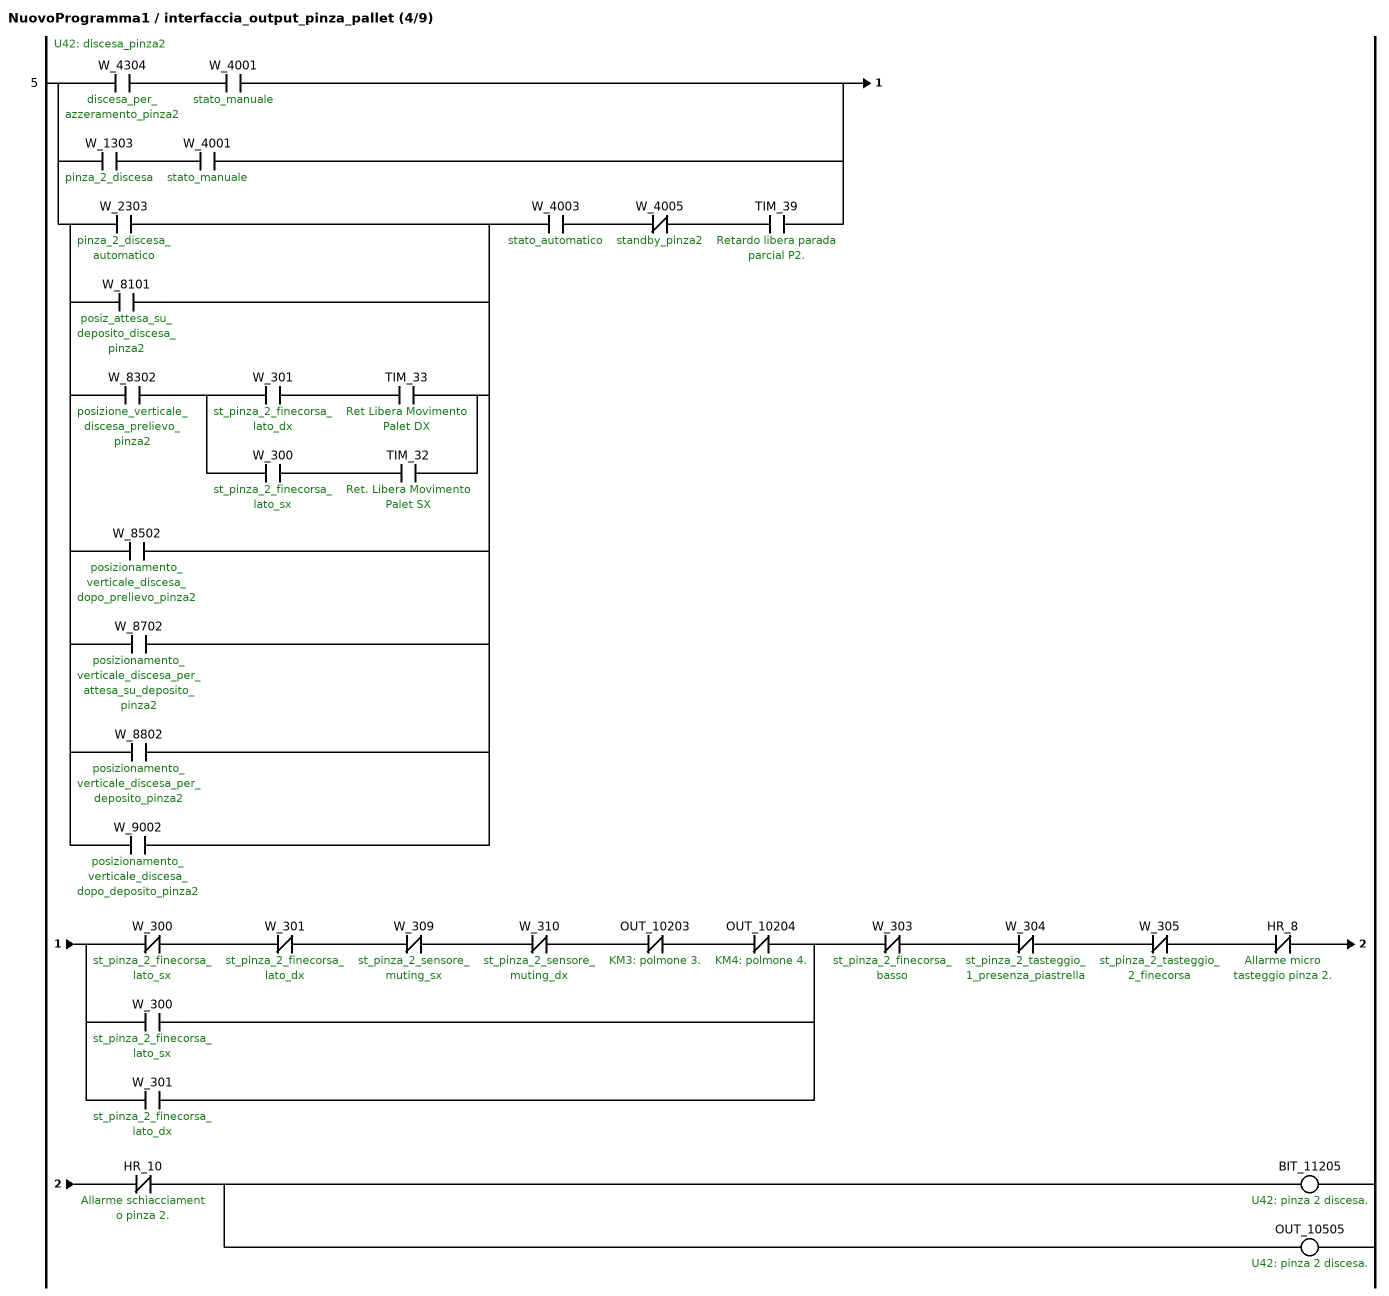
; [picture p24: NuovoProgramma1 / interfaccia_output_pinza_pallet, rungs 5-5]
; rung 5: U42: discesa_pinza2
LD W_4304  ; discesa_per_azzeramento_pinza2
AND W_4001  ; stato_manuale
LD W_1303  ; pinza_2_discesa
AND W_4001  ; stato_manuale
ORLD
LD W_2303  ; pinza_2_discesa_automatico
OR W_8101  ; posiz_attesa_su_deposito_discesa_pinza2
LD W_8302  ; posizione_verticale_discesa_prelievo_pinza2
LD W_301  ; st_pinza_2_finecorsa_lato_dx
AND TIM_33  ; Ret Libera Movimento Palet DX
LD W_300  ; st_pinza_2_finecorsa_lato_sx
AND TIM_32  ; Ret. Libera Movimento Palet SX
ORLD
ANDLD
ORLD
OR W_8502  ; posizionamento_verticale_discesa_dopo_prelievo_pinza2
OR W_8702  ; posizionamento_verticale_discesa_per_attesa_su_deposito_pinza2
OR W_8802  ; posizionamento_verticale_discesa_per_deposito_pinza2
OR W_9002  ; posizionamento_verticale_discesa_dopo_deposito_pinza2
AND W_4003  ; stato_automatico
ANDNOT W_4005  ; standby_pinza2
AND TIM_39  ; Retardo libera parada parcial P2.
ORLD
LDNOT W_300  ; st_pinza_2_finecorsa_lato_sx
ANDNOT W_301  ; st_pinza_2_finecorsa_lato_dx
ANDNOT W_309  ; st_pinza_2_sensore_muting_sx
ANDNOT W_310  ; st_pinza_2_sensore_muting_dx
ANDNOT OUT_10203  ; KM3: polmone 3.
ANDNOT OUT_10204  ; KM4: polmone 4.
OR W_300  ; st_pinza_2_finecorsa_lato_sx
OR W_301  ; st_pinza_2_finecorsa_lato_dx
ANDLD
ANDNOT W_303  ; st_pinza_2_finecorsa_basso
ANDNOT W_304  ; st_pinza_2_tasteggio_1_presenza_piastrella
ANDNOT W_305  ; st_pinza_2_tasteggio_2_finecorsa
ANDNOT HR_8  ; Allarme micro tasteggio pinza 2.
ANDNOT HR_10  ; Allarme schiacciamento pinza 2.
OUT BIT_11205  ; U42: pinza 2 discesa.
OUT OUT_10505  ; U42: pinza 2 discesa.

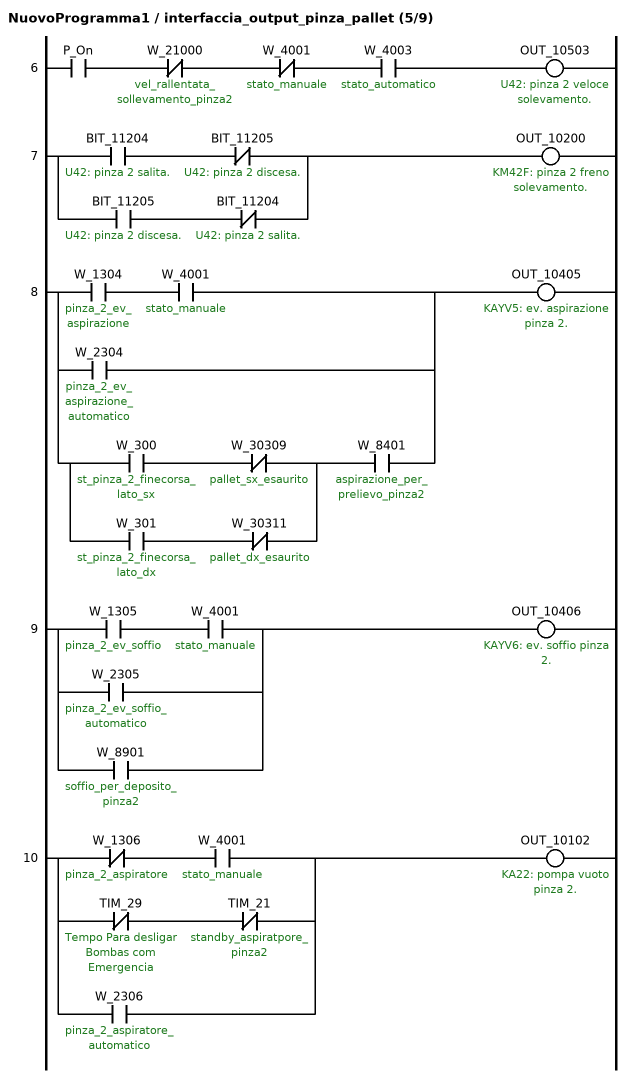
; rung 6
LD P_On
ANDNOT W_21000  ; vel_rallentata_sollevamento_pinza2
ANDNOT W_4001  ; stato_manuale
AND W_4003  ; stato_automatico
OUT OUT_10503  ; U42: pinza 2 veloce solevamento.
; rung 7
LD BIT_11204  ; U42: pinza 2 salita.
ANDNOT BIT_11205  ; U42: pinza 2 discesa.
LD BIT_11205  ; U42: pinza 2 discesa.
ANDNOT BIT_11204  ; U42: pinza 2 salita.
ORLD
OUT OUT_10200  ; KM42F: pinza 2 freno solevamento.
; rung 8
LD W_1304  ; pinza_2_ev_aspirazione
AND W_4001  ; stato_manuale
OR W_2304  ; pinza_2_ev_aspirazione_automatico
LD W_300  ; st_pinza_2_finecorsa_lato_sx
ANDNOT W_30309  ; pallet_sx_esaurito
LD W_301  ; st_pinza_2_finecorsa_lato_dx
ANDNOT W_30311  ; pallet_dx_esaurito
ORLD
AND W_8401  ; aspirazione_per_prelievo_pinza2
ORLD
OUT OUT_10405  ; KAYV5: ev. aspirazione pinza 2.
; rung 9
LD W_1305  ; pinza_2_ev_soffio
AND W_4001  ; stato_manuale
OR W_2305  ; pinza_2_ev_soffio_automatico
OR W_8901  ; soffio_per_deposito_pinza2
OUT OUT_10406  ; KAYV6: ev. soffio pinza 2.
; rung 10
LDNOT W_1306  ; pinza_2_aspiratore
AND W_4001  ; stato_manuale
LDNOT TIM_29  ; Tempo Para desligar Bombas com Emergencia
ANDNOT TIM_21  ; standby_aspiratpore_pinza2
ORLD
OR W_2306  ; pinza_2_aspiratore_automatico
OUT OUT_10102  ; KA22: pompa vuoto pinza 2.

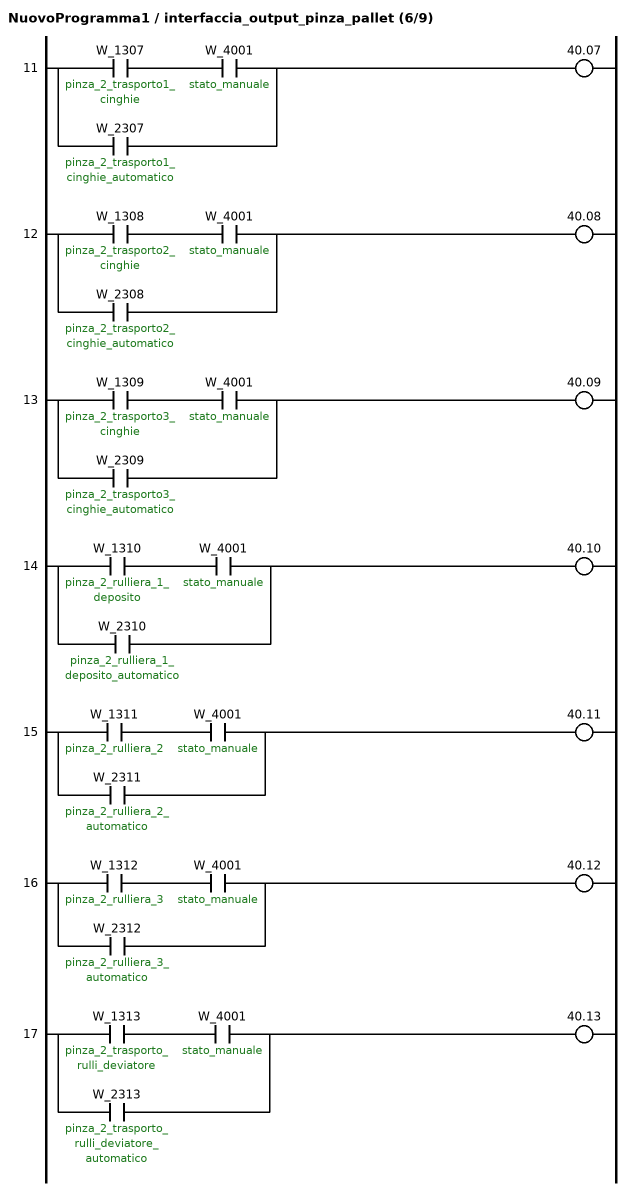
; rung 11
LD W_1307  ; pinza_2_trasporto1_cinghie
AND W_4001  ; stato_manuale
OR W_2307  ; pinza_2_trasporto1_cinghie_automatico
OUT 40.07
; rung 12
LD W_1308  ; pinza_2_trasporto2_cinghie
AND W_4001  ; stato_manuale
OR W_2308  ; pinza_2_trasporto2_cinghie_automatico
OUT 40.08
; rung 13
LD W_1309  ; pinza_2_trasporto3_cinghie
AND W_4001  ; stato_manuale
OR W_2309  ; pinza_2_trasporto3_cinghie_automatico
OUT 40.09
; rung 14
LD W_1310  ; pinza_2_rulliera_1_deposito
AND W_4001  ; stato_manuale
OR W_2310  ; pinza_2_rulliera_1_deposito_automatico
OUT 40.10
; rung 15
LD W_1311  ; pinza_2_rulliera_2
AND W_4001  ; stato_manuale
OR W_2311  ; pinza_2_rulliera_2_automatico
OUT 40.11
; rung 16
LD W_1312  ; pinza_2_rulliera_3
AND W_4001  ; stato_manuale
OR W_2312  ; pinza_2_rulliera_3_automatico
OUT 40.12
; rung 17
LD W_1313  ; pinza_2_trasporto_rulli_deviatore
AND W_4001  ; stato_manuale
OR W_2313  ; pinza_2_trasporto_rulli_deviatore_automatico
OUT 40.13

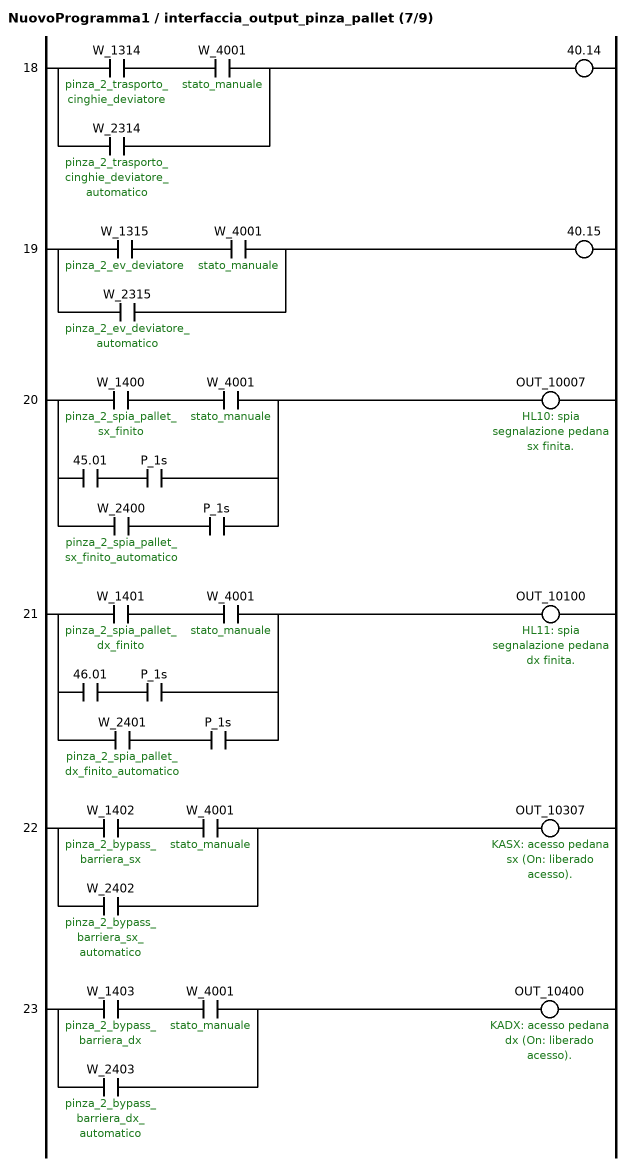
; rung 18
LD W_1314  ; pinza_2_trasporto_cinghie_deviatore
AND W_4001  ; stato_manuale
OR W_2314  ; pinza_2_trasporto_cinghie_deviatore_automatico
OUT 40.14
; rung 19
LD W_1315  ; pinza_2_ev_deviatore
AND W_4001  ; stato_manuale
OR W_2315  ; pinza_2_ev_deviatore_automatico
OUT 40.15
; rung 20
LD W_1400  ; pinza_2_spia_pallet_sx_finito
AND W_4001  ; stato_manuale
LD 45.01
AND P_1s
ORLD
LD W_2400  ; pinza_2_spia_pallet_sx_finito_automatico
AND P_1s
ORLD
OUT OUT_10007  ; HL10: spia segnalazione pedana sx finita.
; rung 21
LD W_1401  ; pinza_2_spia_pallet_dx_finito
AND W_4001  ; stato_manuale
LD 46.01
AND P_1s
ORLD
LD W_2401  ; pinza_2_spia_pallet_dx_finito_automatico
AND P_1s
ORLD
OUT OUT_10100  ; HL11: spia segnalazione pedana dx finita.
; rung 22
LD W_1402  ; pinza_2_bypass_barriera_sx
AND W_4001  ; stato_manuale
OR W_2402  ; pinza_2_bypass_barriera_sx_automatico
OUT OUT_10307  ; KASX: acesso pedana sx (On: liberado acesso).
; rung 23
LD W_1403  ; pinza_2_bypass_barriera_dx
AND W_4001  ; stato_manuale
OR W_2403  ; pinza_2_bypass_barriera_dx_automatico
OUT OUT_10400  ; KADX: acesso pedana dx (On: liberado acesso).

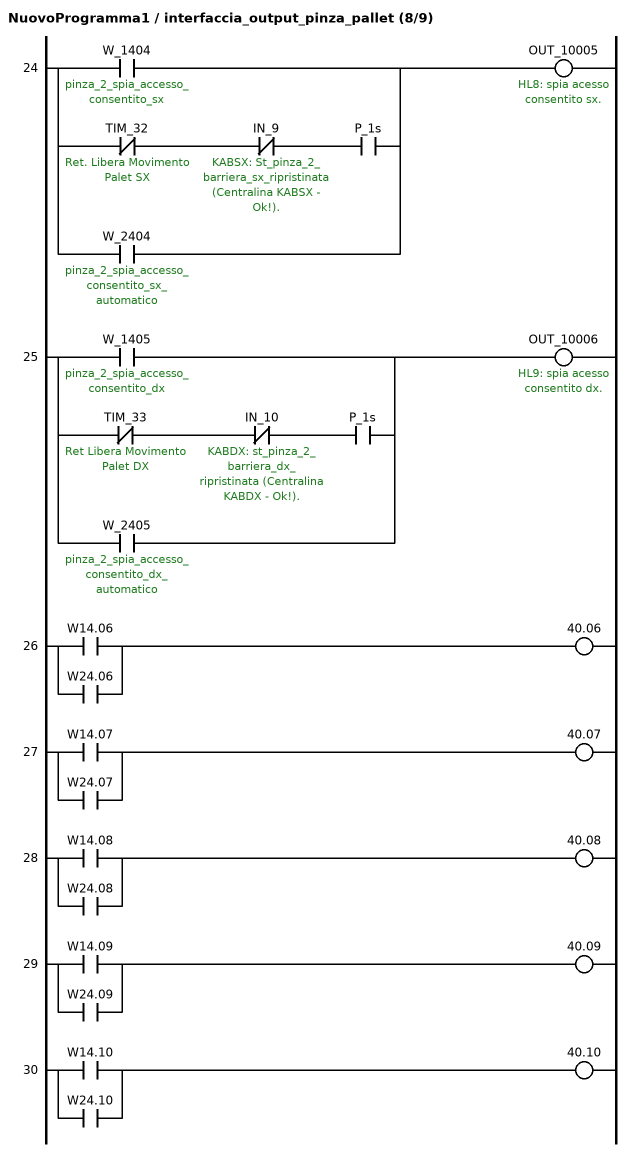
; rung 24
LD W_1404  ; pinza_2_spia_accesso_consentito_sx
LDNOT TIM_32  ; Ret. Libera Movimento Palet SX
ANDNOT IN_9  ; KABSX: St_pinza_2_barriera_sx_ripristinata (Centralina KABSX - Ok!).
AND P_1s
ORLD
OR W_2404  ; pinza_2_spia_accesso_consentito_sx_automatico
OUT OUT_10005  ; HL8: spia acesso consentito sx.
; rung 25
LD W_1405  ; pinza_2_spia_accesso_consentito_dx
LDNOT TIM_33  ; Ret Libera Movimento Palet DX
ANDNOT IN_10  ; KABDX: st_pinza_2_barriera_dx_ripristinata (Centralina KABDX - Ok!).
AND P_1s
ORLD
OR W_2405  ; pinza_2_spia_accesso_consentito_dx_automatico
OUT OUT_10006  ; HL9: spia acesso consentito dx.
; rung 26
LD W14.06
OR W24.06
OUT 40.06
; rung 27
LD W14.07
OR W24.07
OUT 40.07
; rung 28
LD W14.08
OR W24.08
OUT 40.08
; rung 29
LD W14.09
OR W24.09
OUT 40.09
; rung 30
LD W14.10
OR W24.10
OUT 40.10

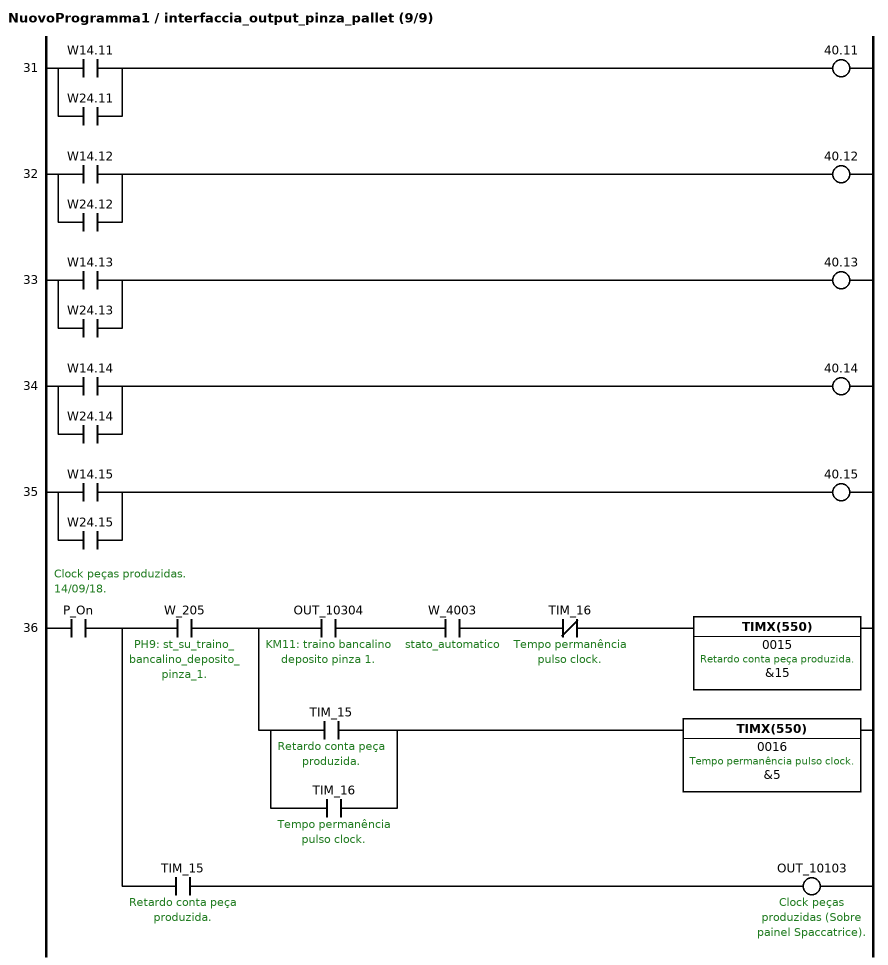
; rung 31
LD W14.11
OR W24.11
OUT 40.11
; rung 32
LD W14.12
OR W24.12
OUT 40.12
; rung 33
LD W14.13
OR W24.13
OUT 40.13
; rung 34
LD W14.14
OR W24.14
OUT 40.14
; rung 35
LD W14.15
OR W24.15
OUT 40.15
; rung 36: Clock peças produzidas. / 14/09/18.
LD P_On
OUT TR0
AND W_205  ; PH9: st_su_traino_bancalino_deposito_pinza_1.
OUT TR1
AND OUT_10304  ; KM11: traino bancalino deposito pinza 1.
AND W_4003  ; stato_automatico
ANDNOT TIM_16  ; Tempo permanência pulso clock.
TIMX(550) 0015 &15  ; Retardo conta peça produzida.
LD TR1
LD TIM_15  ; Retardo conta peça produzida.
OR TIM_16  ; Tempo permanência pulso clock.
ANDLD
TIMX(550) 0016 &5  ; Tempo permanência pulso clock.
LD TR0
AND TIM_15  ; Retardo conta peça produzida.
OUT OUT_10103  ; Clock peças produzidas (Sobre painel Spaccatrice).

### Section manuale

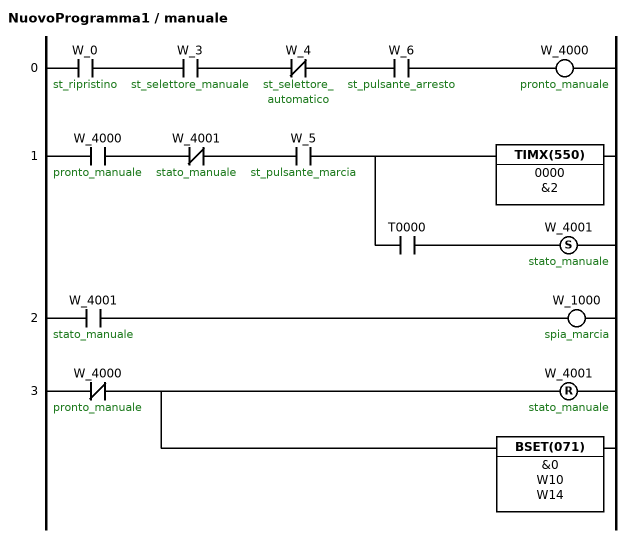
; rung 0
LD W_0  ; st_ripristino
AND W_3  ; st_selettore_manuale
ANDNOT W_4  ; st_selettore_automatico
AND W_6  ; st_pulsante_arresto
OUT W_4000  ; pronto_manuale
; rung 1
LD W_4000  ; pronto_manuale
ANDNOT W_4001  ; stato_manuale
AND W_5  ; st_pulsante_marcia
TIMX(550) 0000 &2
AND T0000
SET W_4001  ; stato_manuale
; rung 2
LD W_4001  ; stato_manuale
OUT W_1000  ; spia_marcia
; rung 3
LDNOT W_4000  ; pronto_manuale
RSET W_4001  ; stato_manuale
BSET(071) &0 W10 W14

### Section abilitazioni

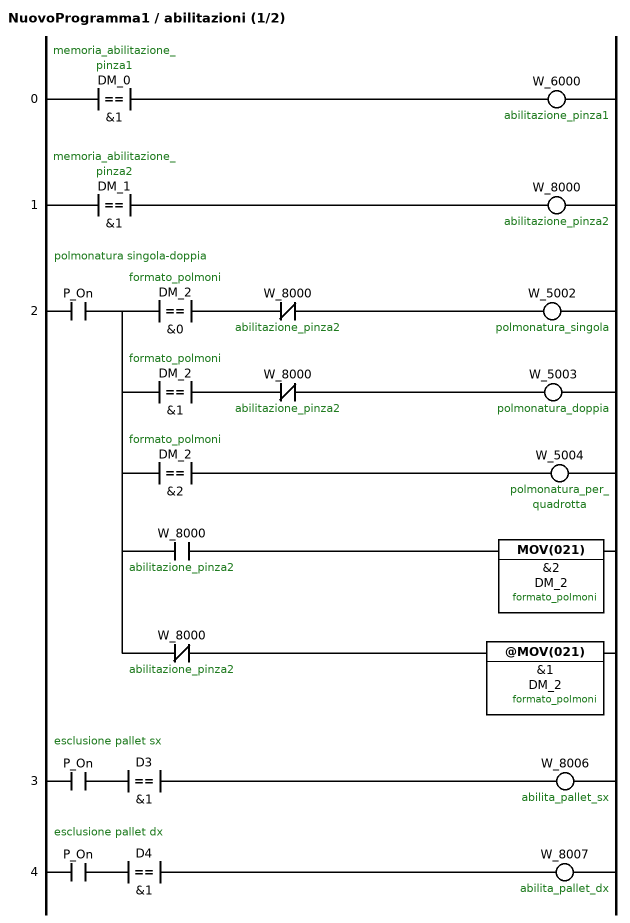
; rung 0
LD=(300) DM_0 &1  ; memoria_abilitazione_pinza1
OUT W_6000  ; abilitazione_pinza1
; rung 1
LD=(300) DM_1 &1  ; memoria_abilitazione_pinza2
OUT W_8000  ; abilitazione_pinza2
; rung 2: polmonatura singola-doppia
LD P_On
OUT TR0
AND=(300) DM_2 &0  ; formato_polmoni
ANDNOT W_8000  ; abilitazione_pinza2
OUT W_5002  ; polmonatura_singola
LD TR0
AND=(300) DM_2 &1  ; formato_polmoni
ANDNOT W_8000  ; abilitazione_pinza2
OUT W_5003  ; polmonatura_doppia
LD TR0
AND=(300) DM_2 &2  ; formato_polmoni
OUT W_5004  ; polmonatura_per_quadrotta
LD TR0
AND W_8000  ; abilitazione_pinza2
MOV(021) &2 DM_2  ; formato_polmoni
LD TR0
ANDNOT W_8000  ; abilitazione_pinza2
@MOV(021) &1 DM_2  ; formato_polmoni
; rung 3: esclusione pallet sx
LD P_On
AND=(300) D3 &1
OUT W_8006  ; abilita_pallet_sx
; rung 4: esclusione pallet dx
LD P_On
AND=(300) D4 &1
OUT W_8007  ; abilita_pallet_dx

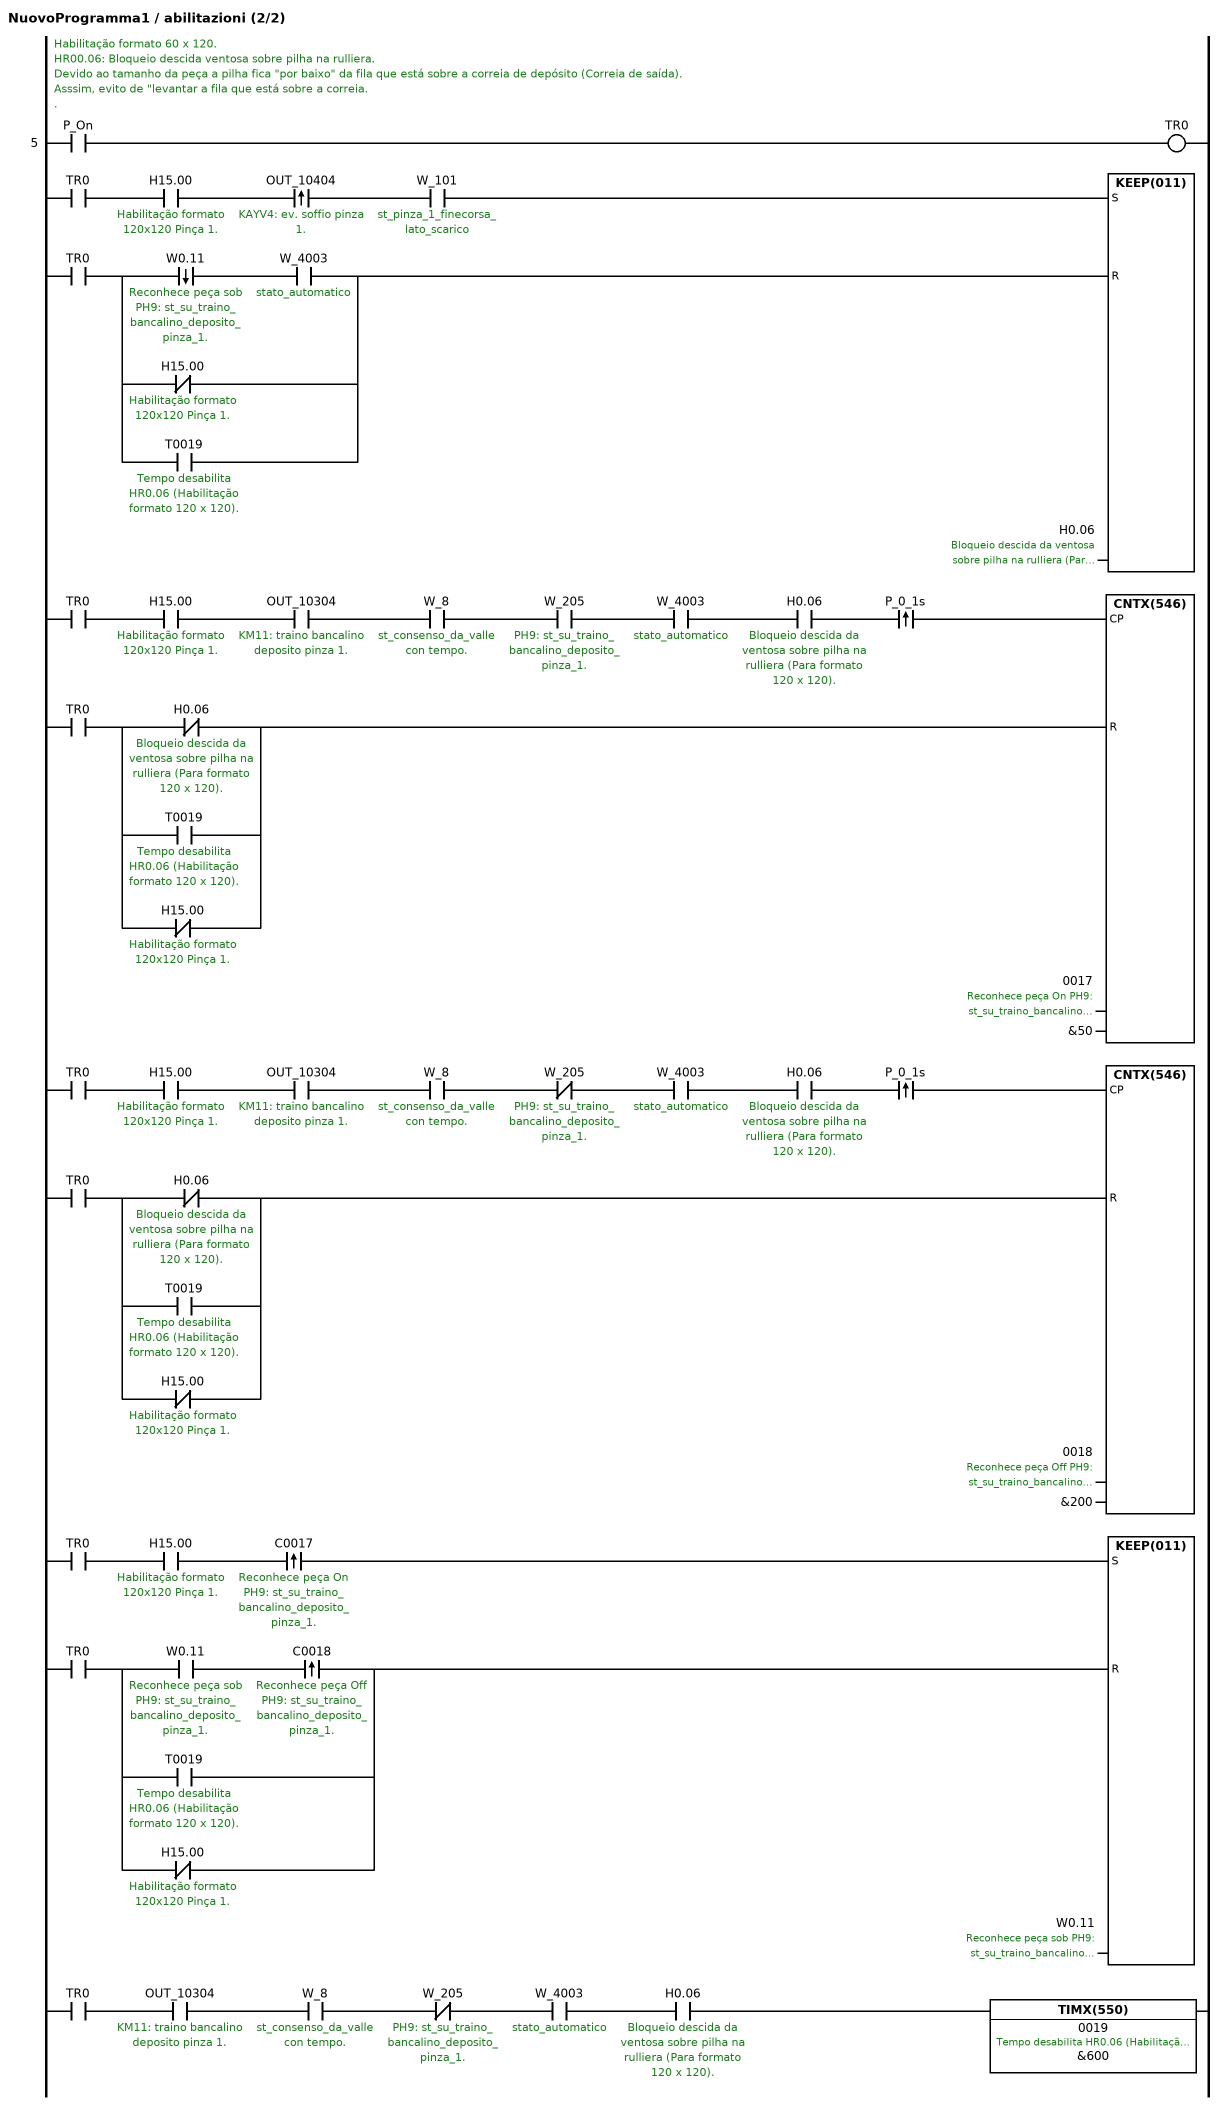
; rung 5: Habilitação formato 60 x 120. / HR00.06: Bloqueio descida ventosa sobre pilha na rulliera. / Devido ao tamanho da peça a pilha fica "por baixo" da fila que está sobre a correia de depósito (Correia de saída). / Asssim, evito de "levantar a fila que está sobre a correia. / .
LD P_On
OUT TR0
AND H15.00  ; Habilitação formato 120x120 Pinça 1.
@AND OUT_10404  ; KAYV4: ev. soffio pinza 1.
AND W_101  ; st_pinza_1_finecorsa_lato_scarico
LD TR0
%LD W0.11  ; Reconhece peça sob PH9: st_su_traino_bancalino_deposito_pinza_1.
AND W_4003  ; stato_automatico
ORNOT H15.00  ; Habilitação formato 120x120 Pinça 1.
OR T0019  ; Tempo desabilita HR0.06 (Habilitação formato 120 x 120).
ANDLD
KEEP(011) H0.06  ; Bloqueio descida da ventosa sobre pilha na rulliera (Para formato 120 x 120).  // On: material depositado sobre correia de saída. / Off: passou peça sob Ftc se saída (IN2.09_PH9: st_su_traino_bancalino_deposito_pinza_1). / .
LD TR0
AND H15.00  ; Habilitação formato 120x120 Pinça 1.
AND OUT_10304  ; KM11: traino bancalino deposito pinza 1.
AND W_8  ; st_consenso_da_valle con tempo.
AND W_205  ; PH9: st_su_traino_bancalino_deposito_pinza_1.
AND W_4003  ; stato_automatico
AND H0.06  ; Bloqueio descida da ventosa sobre pilha na rulliera (Para formato 120 x 120).
@AND P_0_1s
LD TR0
LDNOT H0.06  ; Bloqueio descida da ventosa sobre pilha na rulliera (Para formato 120 x 120).
OR T0019  ; Tempo desabilita HR0.06 (Habilitação formato 120 x 120).
ORNOT H15.00  ; Habilitação formato 120x120 Pinça 1.
ANDLD
CNTX(546) 0017 &50  ; Reconhece peça On PH9: st_su_traino_bancalino_deposito_pinza_1.
LD TR0
AND H15.00  ; Habilitação formato 120x120 Pinça 1.
AND OUT_10304  ; KM11: traino bancalino deposito pinza 1.
AND W_8  ; st_consenso_da_valle con tempo.
ANDNOT W_205  ; PH9: st_su_traino_bancalino_deposito_pinza_1.
AND W_4003  ; stato_automatico
AND H0.06  ; Bloqueio descida da ventosa sobre pilha na rulliera (Para formato 120 x 120).
@AND P_0_1s
LD TR0
LDNOT H0.06  ; Bloqueio descida da ventosa sobre pilha na rulliera (Para formato 120 x 120).
OR T0019  ; Tempo desabilita HR0.06 (Habilitação formato 120 x 120).
ORNOT H15.00  ; Habilitação formato 120x120 Pinça 1.
ANDLD
CNTX(546) 0018 &200  ; Reconhece peça Off PH9: st_su_traino_bancalino_deposito_pinza_1.
LD TR0
AND H15.00  ; Habilitação formato 120x120 Pinça 1.
@AND C0017  ; Reconhece peça On PH9: st_su_traino_bancalino_deposito_pinza_1.
LD TR0
LD W0.11  ; Reconhece peça sob PH9: st_su_traino_bancalino_deposito_pinza_1.
@AND C0018  ; Reconhece peça Off PH9: st_su_traino_bancalino_deposito_pinza_1.
OR T0019  ; Tempo desabilita HR0.06 (Habilitação formato 120 x 120).
ORNOT H15.00  ; Habilitação formato 120x120 Pinça 1.
ANDLD
KEEP(011) W0.11  ; Reconhece peça sob PH9: st_su_traino_bancalino_deposito_pinza_1.
LD TR0
AND OUT_10304  ; KM11: traino bancalino deposito pinza 1.
AND W_8  ; st_consenso_da_valle con tempo.
ANDNOT W_205  ; PH9: st_su_traino_bancalino_deposito_pinza_1.
AND W_4003  ; stato_automatico
AND H0.06  ; Bloqueio descida da ventosa sobre pilha na rulliera (Para formato 120 x 120).
TIMX(550) 0019 &600  ; Tempo desabilita HR0.06 (Habilitação formato 120 x 120).  // Tempo de segurança para o caso de faltar material na linha (E, assim, não acionar a ftc. que reconhece passagem da peça). / .

### Section azzeramento_assi_pinza_ribaltino

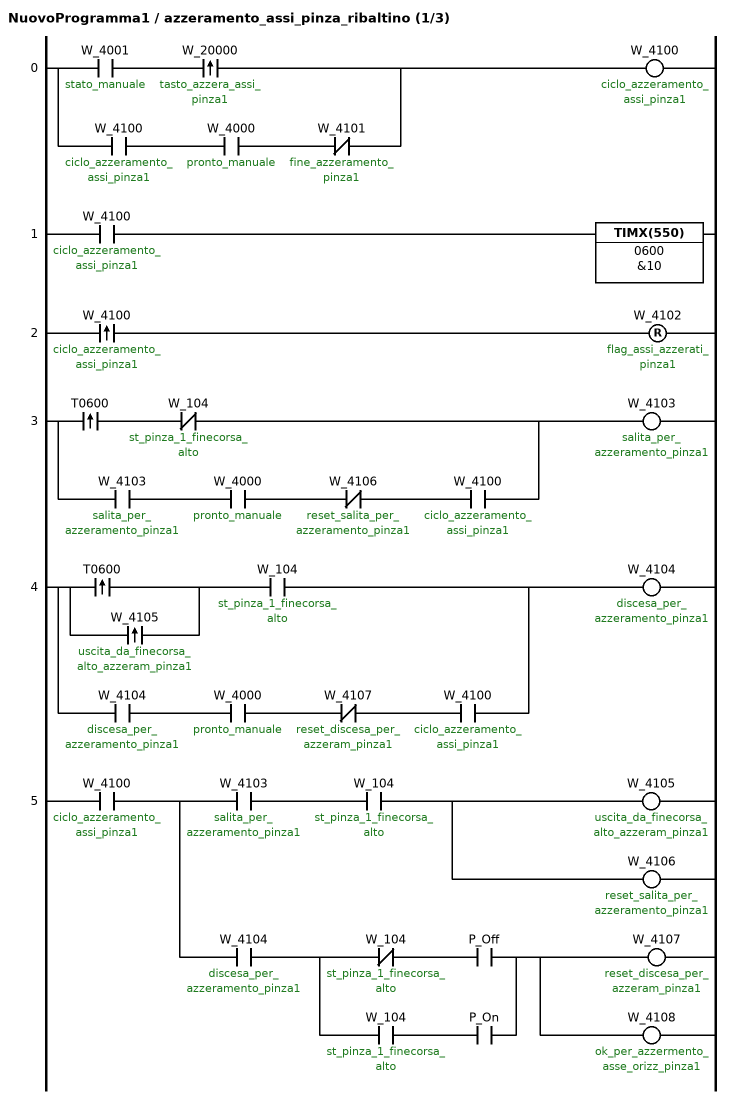
; rung 0
LD W_4001  ; stato_manuale
@AND W_20000  ; tasto_azzera_assi_pinza1
LD W_4100  ; ciclo_azzeramento_assi_pinza1
AND W_4000  ; pronto_manuale
ANDNOT W_4101  ; fine_azzeramento_pinza1
ORLD
OUT W_4100  ; ciclo_azzeramento_assi_pinza1
; rung 1
LD W_4100  ; ciclo_azzeramento_assi_pinza1
TIMX(550) 0600 &10
; rung 2
@LD W_4100  ; ciclo_azzeramento_assi_pinza1
RSET W_4102  ; flag_assi_azzerati_pinza1
; rung 3
@LD T0600
ANDNOT W_104  ; st_pinza_1_finecorsa_alto
LD W_4103  ; salita_per_azzeramento_pinza1
AND W_4000  ; pronto_manuale
ANDNOT W_4106  ; reset_salita_per_azzeramento_pinza1
AND W_4100  ; ciclo_azzeramento_assi_pinza1
ORLD
OUT W_4103  ; salita_per_azzeramento_pinza1
; rung 4
@LD T0600
@OR W_4105  ; uscita_da_finecorsa_alto_azzeram_pinza1
AND W_104  ; st_pinza_1_finecorsa_alto
LD W_4104  ; discesa_per_azzeramento_pinza1
AND W_4000  ; pronto_manuale
ANDNOT W_4107  ; reset_discesa_per_azzeram_pinza1
AND W_4100  ; ciclo_azzeramento_assi_pinza1
ORLD
OUT W_4104  ; discesa_per_azzeramento_pinza1
; rung 5
LD W_4100  ; ciclo_azzeramento_assi_pinza1
OUT TR0
AND W_4103  ; salita_per_azzeramento_pinza1
AND W_104  ; st_pinza_1_finecorsa_alto
OUT W_4105  ; uscita_da_finecorsa_alto_azzeram_pinza1
OUT W_4106  ; reset_salita_per_azzeramento_pinza1
LD TR0
AND W_4104  ; discesa_per_azzeramento_pinza1
LDNOT W_104  ; st_pinza_1_finecorsa_alto
AND P_Off
LD W_104  ; st_pinza_1_finecorsa_alto
AND P_On
ORLD
ANDLD
OUT W_4107  ; reset_discesa_per_azzeram_pinza1
OUT W_4108  ; ok_per_azzermento_asse_orizz_pinza1

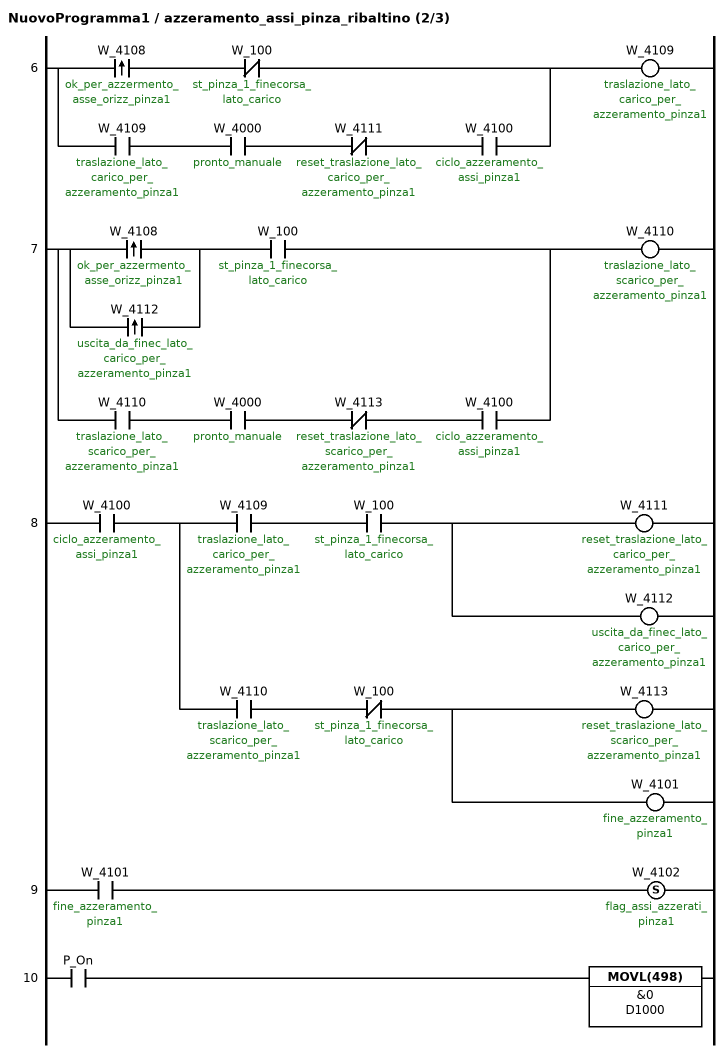
; rung 6
@LD W_4108  ; ok_per_azzermento_asse_orizz_pinza1
ANDNOT W_100  ; st_pinza_1_finecorsa_lato_carico
LD W_4109  ; traslazione_lato_carico_per_azzeramento_pinza1
AND W_4000  ; pronto_manuale
ANDNOT W_4111  ; reset_traslazione_lato_carico_per_azzeramento_pinza1
AND W_4100  ; ciclo_azzeramento_assi_pinza1
ORLD
OUT W_4109  ; traslazione_lato_carico_per_azzeramento_pinza1
; rung 7
@LD W_4108  ; ok_per_azzermento_asse_orizz_pinza1
@OR W_4112  ; uscita_da_finec_lato_carico_per_azzeramento_pinza1
AND W_100  ; st_pinza_1_finecorsa_lato_carico
LD W_4110  ; traslazione_lato_scarico_per_azzeramento_pinza1
AND W_4000  ; pronto_manuale
ANDNOT W_4113  ; reset_traslazione_lato_scarico_per_azzeramento_pinza1
AND W_4100  ; ciclo_azzeramento_assi_pinza1
ORLD
OUT W_4110  ; traslazione_lato_scarico_per_azzeramento_pinza1
; rung 8
LD W_4100  ; ciclo_azzeramento_assi_pinza1
OUT TR0
AND W_4109  ; traslazione_lato_carico_per_azzeramento_pinza1
AND W_100  ; st_pinza_1_finecorsa_lato_carico
OUT W_4111  ; reset_traslazione_lato_carico_per_azzeramento_pinza1
OUT W_4112  ; uscita_da_finec_lato_carico_per_azzeramento_pinza1
LD TR0
AND W_4110  ; traslazione_lato_scarico_per_azzeramento_pinza1
ANDNOT W_100  ; st_pinza_1_finecorsa_lato_carico
OUT W_4113  ; reset_traslazione_lato_scarico_per_azzeramento_pinza1
OUT W_4101  ; fine_azzeramento_pinza1
; rung 9
LD W_4101  ; fine_azzeramento_pinza1
SET W_4102  ; flag_assi_azzerati_pinza1
; rung 10
LD P_On
MOVL(498) &0 D1000

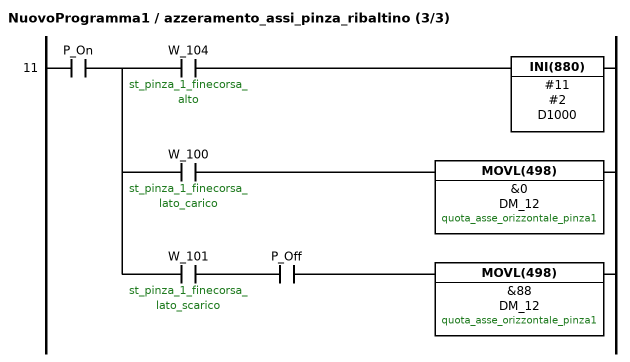
; rung 11
LD P_On
OUT TR0
AND W_104  ; st_pinza_1_finecorsa_alto
INI(880) #11 #2 D1000
LD TR0
AND W_100  ; st_pinza_1_finecorsa_lato_carico
MOVL(498) &0 DM_12  ; quota_asse_orizzontale_pinza1
LD TR0
AND W_101  ; st_pinza_1_finecorsa_lato_scarico
AND P_Off
MOVL(498) &88 DM_12  ; quota_asse_orizzontale_pinza1

### Section azzeramento_assi_pinza_pallet

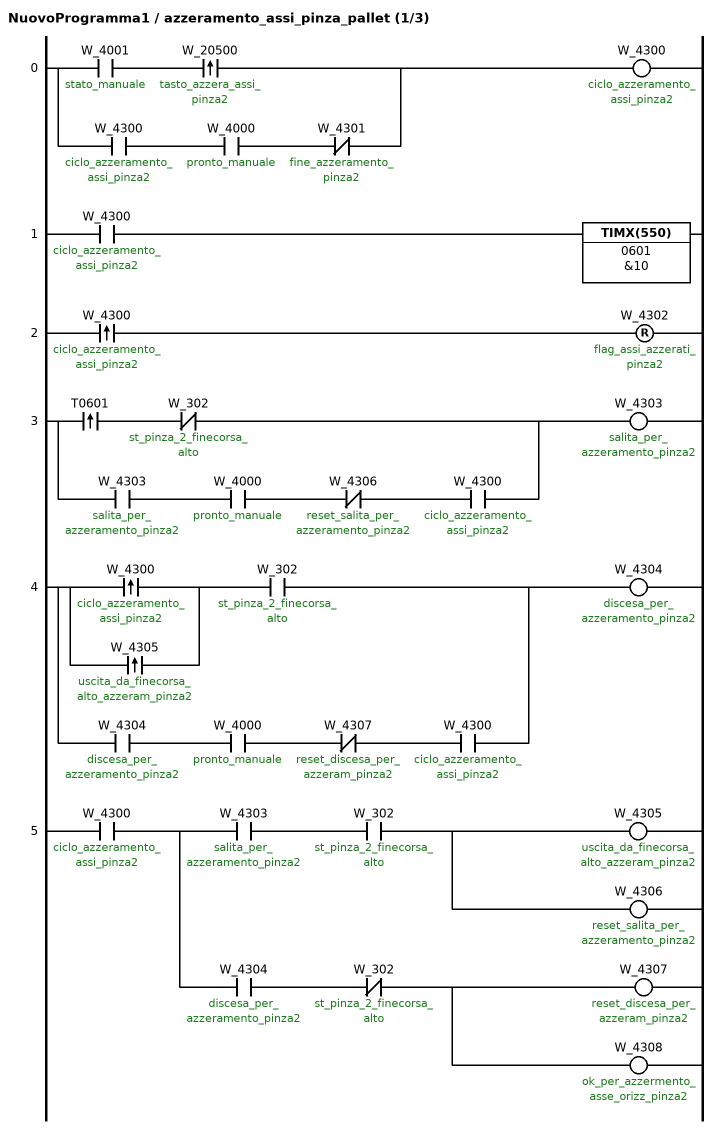
; rung 0
LD W_4001  ; stato_manuale
@AND W_20500  ; tasto_azzera_assi_pinza2
LD W_4300  ; ciclo_azzeramento_assi_pinza2
AND W_4000  ; pronto_manuale
ANDNOT W_4301  ; fine_azzeramento_pinza2
ORLD
OUT W_4300  ; ciclo_azzeramento_assi_pinza2
; rung 1
LD W_4300  ; ciclo_azzeramento_assi_pinza2
TIMX(550) 0601 &10
; rung 2
@LD W_4300  ; ciclo_azzeramento_assi_pinza2
RSET W_4302  ; flag_assi_azzerati_pinza2
; rung 3
@LD T0601
ANDNOT W_302  ; st_pinza_2_finecorsa_alto
LD W_4303  ; salita_per_azzeramento_pinza2
AND W_4000  ; pronto_manuale
ANDNOT W_4306  ; reset_salita_per_azzeramento_pinza2
AND W_4300  ; ciclo_azzeramento_assi_pinza2
ORLD
OUT W_4303  ; salita_per_azzeramento_pinza2
; rung 4
@LD W_4300  ; ciclo_azzeramento_assi_pinza2
@OR W_4305  ; uscita_da_finecorsa_alto_azzeram_pinza2
AND W_302  ; st_pinza_2_finecorsa_alto
LD W_4304  ; discesa_per_azzeramento_pinza2
AND W_4000  ; pronto_manuale
ANDNOT W_4307  ; reset_discesa_per_azzeram_pinza2
AND W_4300  ; ciclo_azzeramento_assi_pinza2
ORLD
OUT W_4304  ; discesa_per_azzeramento_pinza2
; rung 5
LD W_4300  ; ciclo_azzeramento_assi_pinza2
OUT TR0
AND W_4303  ; salita_per_azzeramento_pinza2
AND W_302  ; st_pinza_2_finecorsa_alto
OUT W_4305  ; uscita_da_finecorsa_alto_azzeram_pinza2
OUT W_4306  ; reset_salita_per_azzeramento_pinza2
LD TR0
AND W_4304  ; discesa_per_azzeramento_pinza2
ANDNOT W_302  ; st_pinza_2_finecorsa_alto
OUT W_4307  ; reset_discesa_per_azzeram_pinza2
OUT W_4308  ; ok_per_azzermento_asse_orizz_pinza2

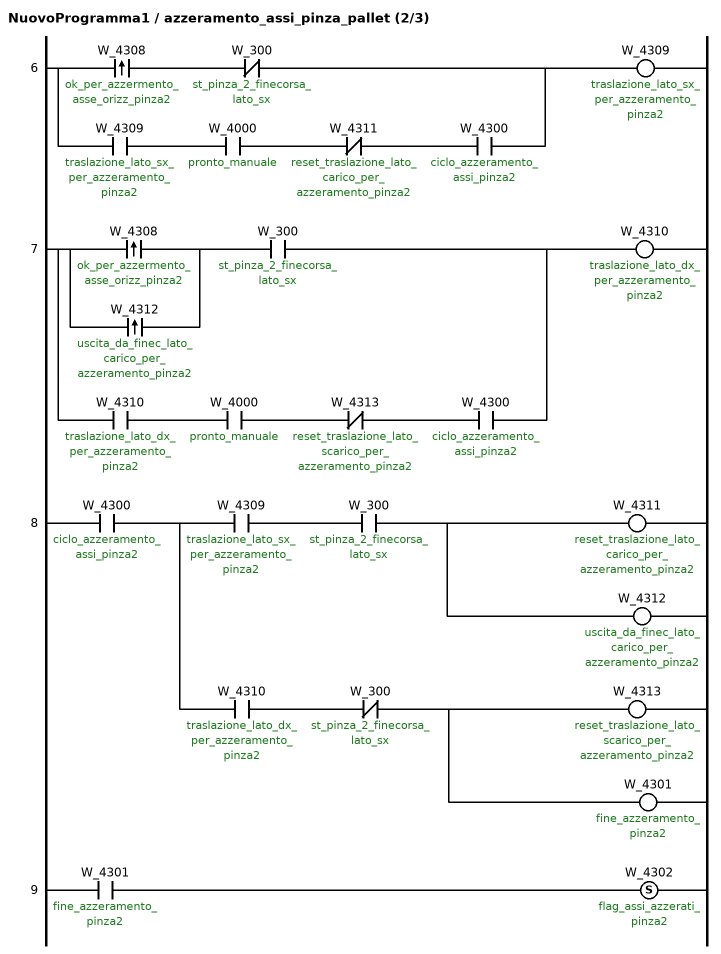
; rung 6
@LD W_4308  ; ok_per_azzermento_asse_orizz_pinza2
ANDNOT W_300  ; st_pinza_2_finecorsa_lato_sx
LD W_4309  ; traslazione_lato_sx_per_azzeramento_pinza2
AND W_4000  ; pronto_manuale
ANDNOT W_4311  ; reset_traslazione_lato_carico_per_azzeramento_pinza2
AND W_4300  ; ciclo_azzeramento_assi_pinza2
ORLD
OUT W_4309  ; traslazione_lato_sx_per_azzeramento_pinza2
; rung 7
@LD W_4308  ; ok_per_azzermento_asse_orizz_pinza2
@OR W_4312  ; uscita_da_finec_lato_carico_per_azzeramento_pinza2
AND W_300  ; st_pinza_2_finecorsa_lato_sx
LD W_4310  ; traslazione_lato_dx_per_azzeramento_pinza2
AND W_4000  ; pronto_manuale
ANDNOT W_4313  ; reset_traslazione_lato_scarico_per_azzeramento_pinza2
AND W_4300  ; ciclo_azzeramento_assi_pinza2
ORLD
OUT W_4310  ; traslazione_lato_dx_per_azzeramento_pinza2
; rung 8
LD W_4300  ; ciclo_azzeramento_assi_pinza2
OUT TR0
AND W_4309  ; traslazione_lato_sx_per_azzeramento_pinza2
AND W_300  ; st_pinza_2_finecorsa_lato_sx
OUT W_4311  ; reset_traslazione_lato_carico_per_azzeramento_pinza2
OUT W_4312  ; uscita_da_finec_lato_carico_per_azzeramento_pinza2
LD TR0
AND W_4310  ; traslazione_lato_dx_per_azzeramento_pinza2
ANDNOT W_300  ; st_pinza_2_finecorsa_lato_sx
OUT W_4313  ; reset_traslazione_lato_scarico_per_azzeramento_pinza2
OUT W_4301  ; fine_azzeramento_pinza2
; rung 9
LD W_4301  ; fine_azzeramento_pinza2
SET W_4302  ; flag_assi_azzerati_pinza2

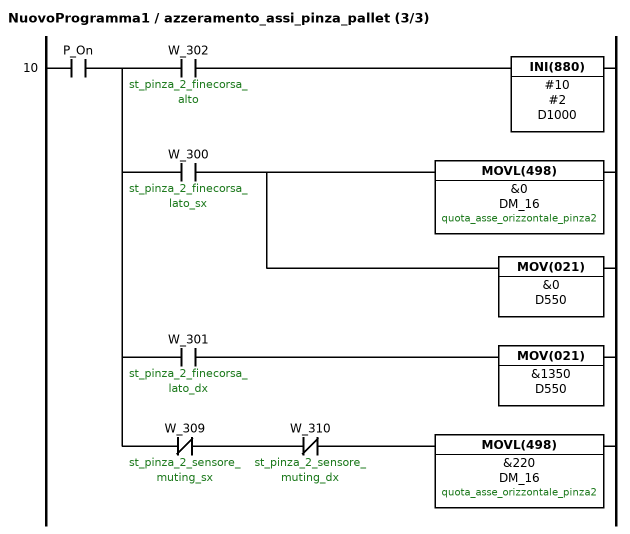
; rung 10
LD P_On
OUT TR0
AND W_302  ; st_pinza_2_finecorsa_alto
INI(880) #10 #2 D1000
LD TR0
AND W_300  ; st_pinza_2_finecorsa_lato_sx
MOVL(498) &0 DM_16  ; quota_asse_orizzontale_pinza2
MOV(021) &0 D550
LD TR0
AND W_301  ; st_pinza_2_finecorsa_lato_dx
MOV(021) &1350 D550
LD TR0
ANDNOT W_309  ; st_pinza_2_sensore_muting_sx
ANDNOT W_310  ; st_pinza_2_sensore_muting_dx
MOVL(498) &220 DM_16  ; quota_asse_orizzontale_pinza2

### Section automatico_generale

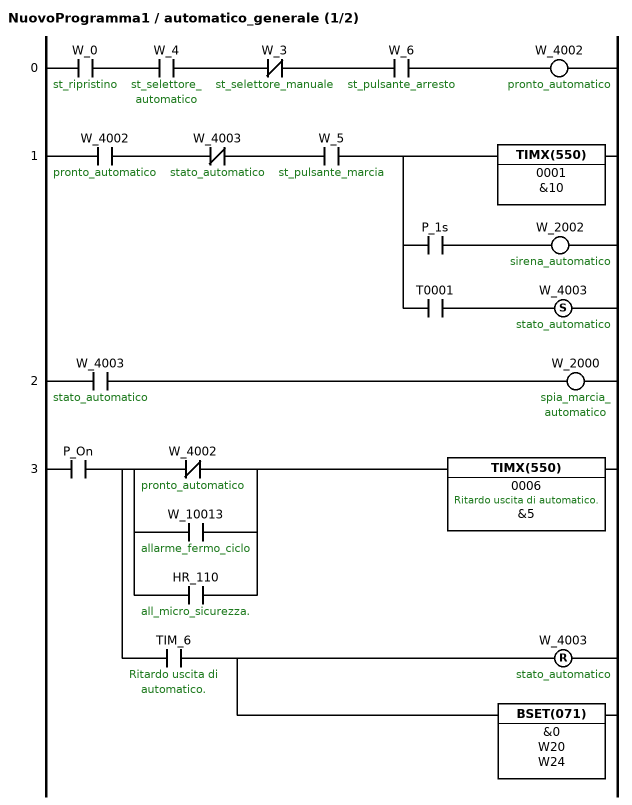
; rung 0
LD W_0  ; st_ripristino
AND W_4  ; st_selettore_automatico
ANDNOT W_3  ; st_selettore_manuale
AND W_6  ; st_pulsante_arresto
OUT W_4002  ; pronto_automatico
; rung 1
LD W_4002  ; pronto_automatico
ANDNOT W_4003  ; stato_automatico
AND W_5  ; st_pulsante_marcia
OUT TR0
TIMX(550) 0001 &10
AND P_1s
OUT W_2002  ; sirena_automatico
LD TR0
AND T0001
SET W_4003  ; stato_automatico
; rung 2
LD W_4003  ; stato_automatico
OUT W_2000  ; spia_marcia_automatico
; rung 3
LD P_On
OUT TR0
LDNOT W_4002  ; pronto_automatico
OR W_10013  ; allarme_fermo_ciclo
OR HR_110  ; all_micro_sicurezza.
ANDLD
TIMX(550) 0006 &5  ; Ritardo uscita di automatico.
LD TR0
AND TIM_6  ; Ritardo uscita di automatico.
RSET W_4003  ; stato_automatico
BSET(071) &0 W20 W24

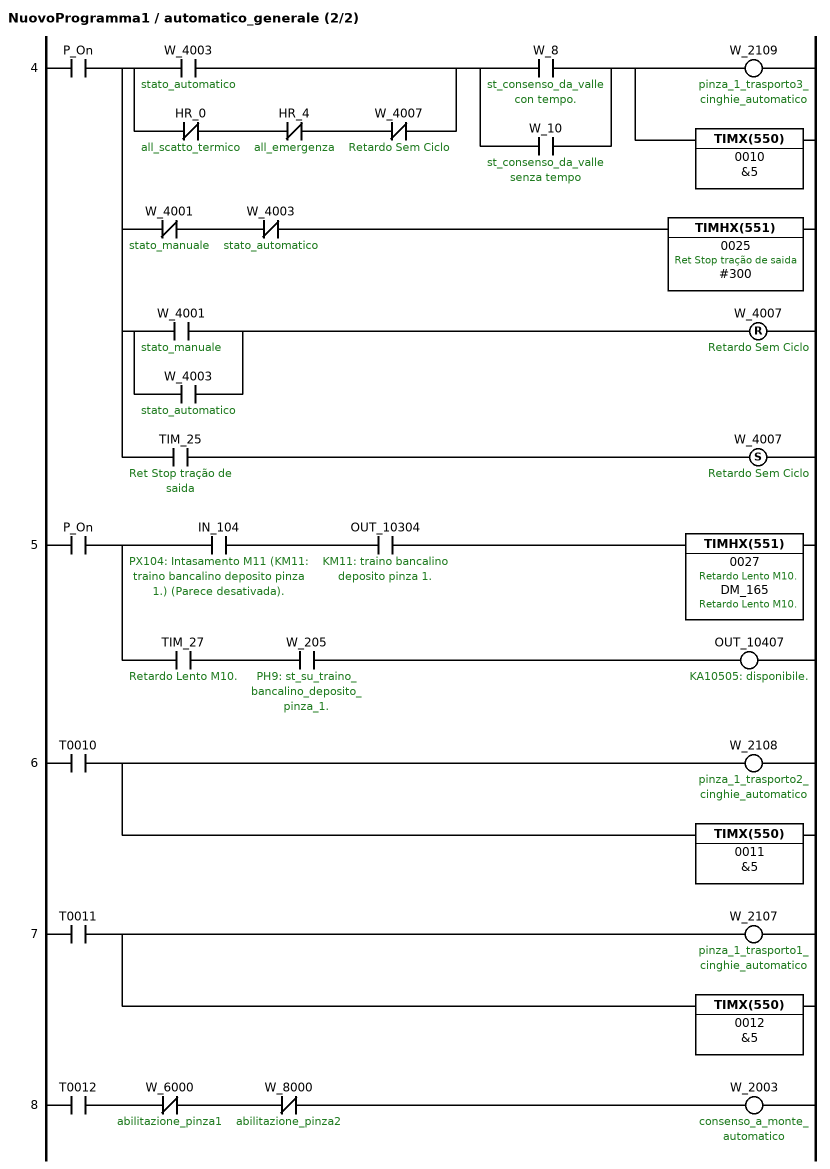
; rung 4
LD P_On
OUT TR0
LD W_4003  ; stato_automatico
LDNOT HR_0  ; all_scatto_termico
ANDNOT HR_4  ; all_emergenza
ANDNOT W_4007  ; Retardo Sem Ciclo
ORLD
ANDLD
LD W_8  ; st_consenso_da_valle con tempo.
OR W_10  ; st_consenso_da_valle senza tempo
ANDLD
OUT W_2109  ; pinza_1_trasporto3_cinghie_automatico
TIMX(550) 0010 &5
LD TR0
ANDNOT W_4001  ; stato_manuale
ANDNOT W_4003  ; stato_automatico
TIMHX(551) 0025 #300  ; Ret Stop tração de saida
LD TR0
LD W_4001  ; stato_manuale
OR W_4003  ; stato_automatico
ANDLD
RSET W_4007  ; Retardo Sem Ciclo
LD TR0
AND TIM_25  ; Ret Stop tração de saida
SET W_4007  ; Retardo Sem Ciclo
; rung 5
LD P_On
OUT TR0
AND IN_104  ; PX104: Intasamento M11 (KM11: traino bancalino deposito pinza 1.) (Parece desativada).
AND OUT_10304  ; KM11: traino bancalino deposito pinza 1.
TIMHX(551) 0027 DM_165  ; Retardo Lento M10.
LD TR0
AND TIM_27  ; Retardo Lento M10.
AND W_205  ; PH9: st_su_traino_bancalino_deposito_pinza_1.
OUT OUT_10407  ; KA10505: disponibile.
; rung 6
LD T0010
OUT W_2108  ; pinza_1_trasporto2_cinghie_automatico
TIMX(550) 0011 &5
; rung 7
LD T0011
OUT W_2107  ; pinza_1_trasporto1_cinghie_automatico
TIMX(550) 0012 &5
; rung 8
LD T0012
ANDNOT W_6000  ; abilitazione_pinza1
ANDNOT W_8000  ; abilitazione_pinza2
OUT W_2003  ; consenso_a_monte_automatico

### Section automatico_pinza_ribaltino

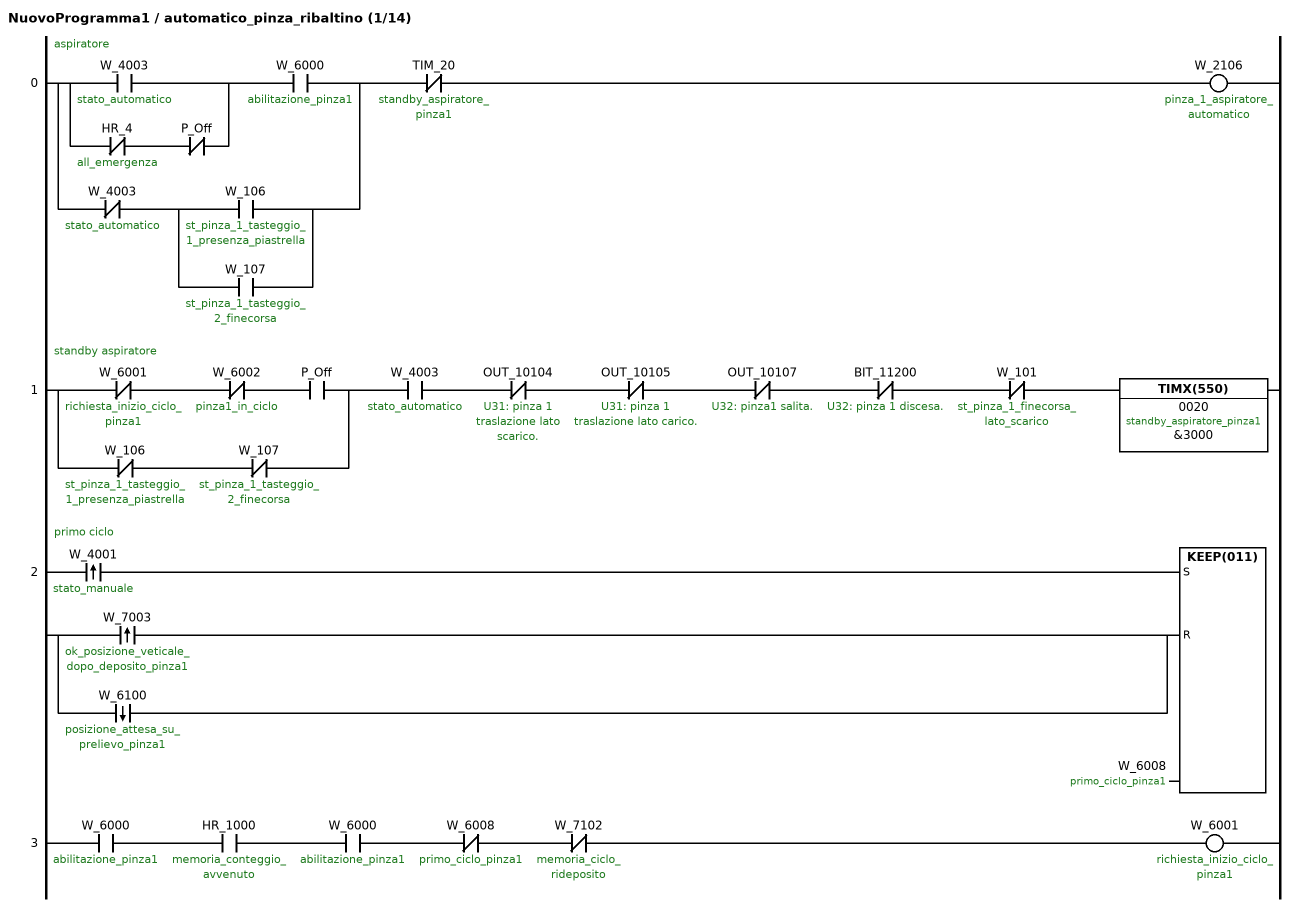
; rung 0: aspiratore
LD W_4003  ; stato_automatico
LDNOT HR_4  ; all_emergenza
ANDNOT P_Off
ORLD
AND W_6000  ; abilitazione_pinza1
LDNOT W_4003  ; stato_automatico
LD W_106  ; st_pinza_1_tasteggio_1_presenza_piastrella
OR W_107  ; st_pinza_1_tasteggio_2_finecorsa
ANDLD
ORLD
ANDNOT TIM_20  ; standby_aspiratore_pinza1
OUT W_2106  ; pinza_1_aspiratore_automatico
; rung 1: standby aspiratore
LDNOT W_6001  ; richiesta_inizio_ciclo_pinza1
ANDNOT W_6002  ; pinza1_in_ciclo
AND P_Off
LDNOT W_106  ; st_pinza_1_tasteggio_1_presenza_piastrella
ANDNOT W_107  ; st_pinza_1_tasteggio_2_finecorsa
ORLD
AND W_4003  ; stato_automatico
ANDNOT OUT_10104  ; U31: pinza 1 traslazione lato scarico.
ANDNOT OUT_10105  ; U31: pinza 1 traslazione lato carico.
ANDNOT OUT_10107  ; U32: pinza1 salita.
ANDNOT BIT_11200  ; U32: pinza 1 discesa.
ANDNOT W_101  ; st_pinza_1_finecorsa_lato_scarico
TIMX(550) 0020 &3000  ; standby_aspiratore_pinza1
; rung 2: primo ciclo
@LD W_4001  ; stato_manuale
@LD W_7003  ; ok_posizione_veticale_dopo_deposito_pinza1
%OR W_6100  ; posizione_attesa_su_prelievo_pinza1
KEEP(011) W_6008  ; primo_ciclo_pinza1
; rung 3
LD W_6000  ; abilitazione_pinza1
AND HR_1000  ; memoria_conteggio_avvenuto
AND W_6000  ; abilitazione_pinza1
ANDNOT W_6008  ; primo_ciclo_pinza1
ANDNOT W_7102  ; memoria_ciclo_rideposito
OUT W_6001  ; richiesta_inizio_ciclo_pinza1

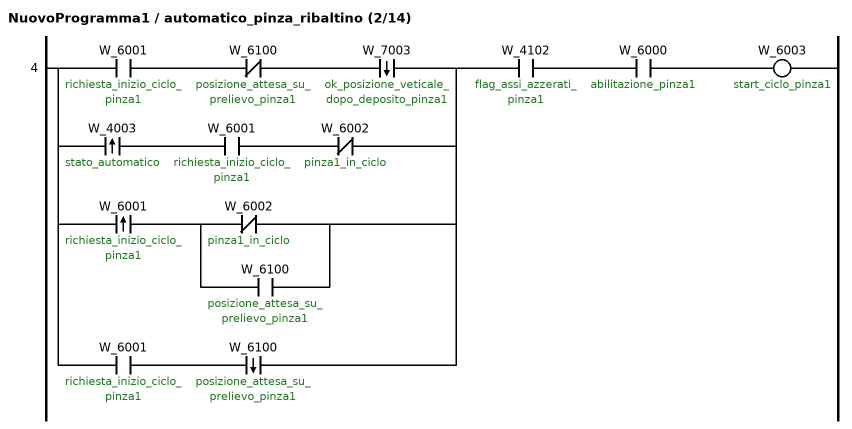
; rung 4
LD W_6001  ; richiesta_inizio_ciclo_pinza1
ANDNOT W_6100  ; posizione_attesa_su_prelievo_pinza1
%AND W_7003  ; ok_posizione_veticale_dopo_deposito_pinza1
@LD W_4003  ; stato_automatico
AND W_6001  ; richiesta_inizio_ciclo_pinza1
ANDNOT W_6002  ; pinza1_in_ciclo
ORLD
@LD W_6001  ; richiesta_inizio_ciclo_pinza1
LDNOT W_6002  ; pinza1_in_ciclo
OR W_6100  ; posizione_attesa_su_prelievo_pinza1
ANDLD
ORLD
LD W_6001  ; richiesta_inizio_ciclo_pinza1
%AND W_6100  ; posizione_attesa_su_prelievo_pinza1
ORLD
AND W_4102  ; flag_assi_azzerati_pinza1
AND W_6000  ; abilitazione_pinza1
OUT W_6003  ; start_ciclo_pinza1

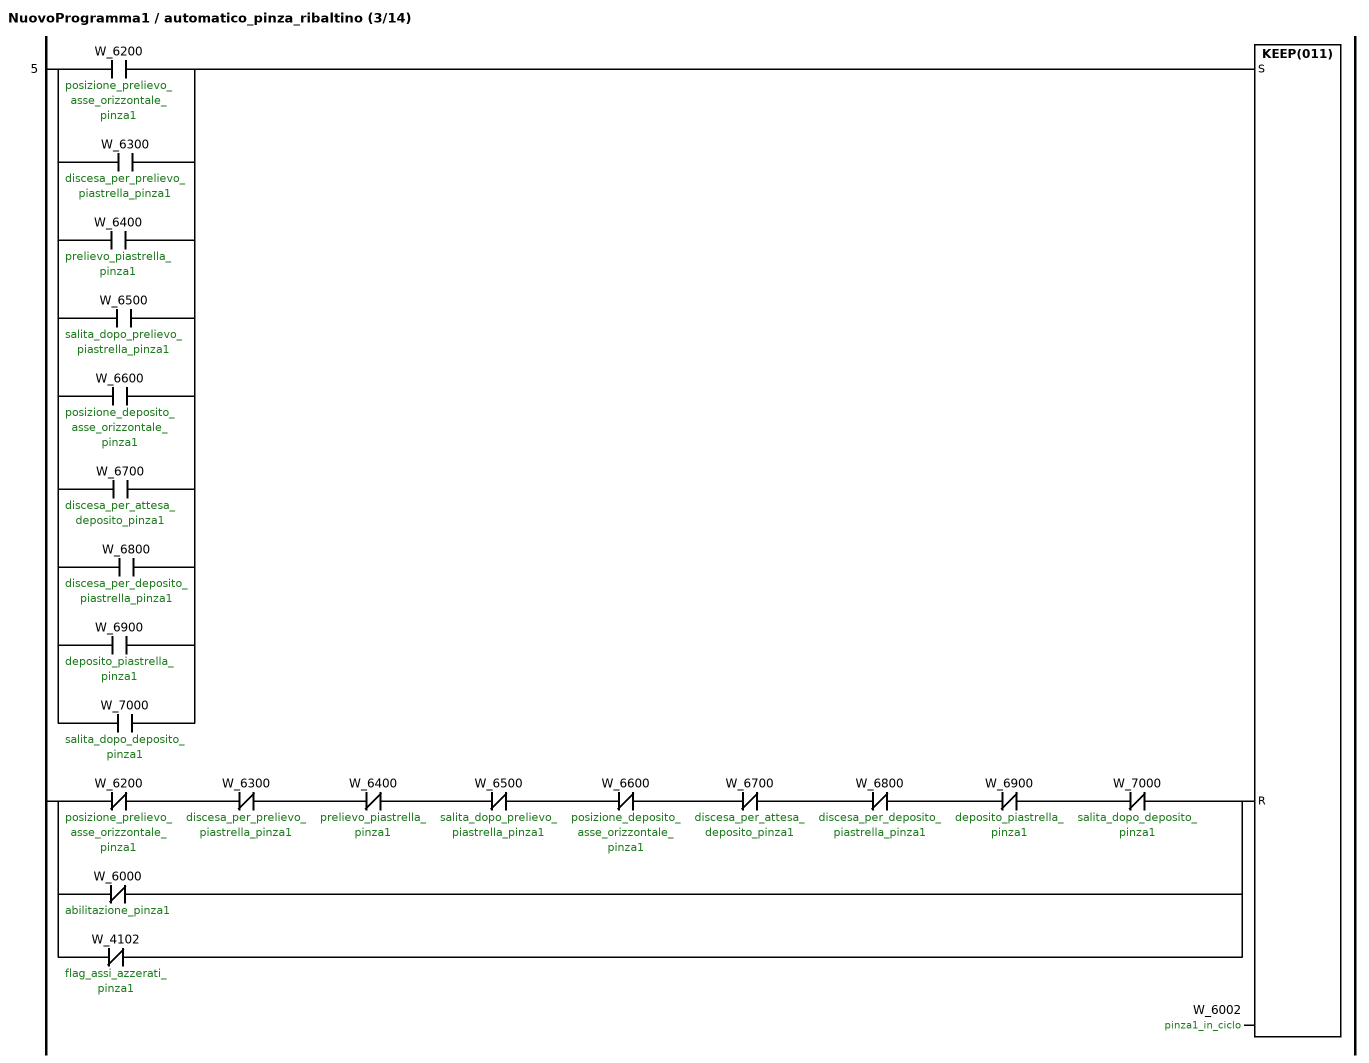
; rung 5
LD W_6200  ; posizione_prelievo_asse_orizzontale_pinza1
OR W_6300  ; discesa_per_prelievo_piastrella_pinza1
OR W_6400  ; prelievo_piastrella_pinza1
OR W_6500  ; salita_dopo_prelievo_piastrella_pinza1
OR W_6600  ; posizione_deposito_asse_orizzontale_pinza1
OR W_6700  ; discesa_per_attesa_deposito_pinza1
OR W_6800  ; discesa_per_deposito_piastrella_pinza1
OR W_6900  ; deposito_piastrella_pinza1
OR W_7000  ; salita_dopo_deposito_pinza1
LDNOT W_6200  ; posizione_prelievo_asse_orizzontale_pinza1
ANDNOT W_6300  ; discesa_per_prelievo_piastrella_pinza1
ANDNOT W_6400  ; prelievo_piastrella_pinza1
ANDNOT W_6500  ; salita_dopo_prelievo_piastrella_pinza1
ANDNOT W_6600  ; posizione_deposito_asse_orizzontale_pinza1
ANDNOT W_6700  ; discesa_per_attesa_deposito_pinza1
ANDNOT W_6800  ; discesa_per_deposito_piastrella_pinza1
ANDNOT W_6900  ; deposito_piastrella_pinza1
ANDNOT W_7000  ; salita_dopo_deposito_pinza1
ORNOT W_6000  ; abilitazione_pinza1
ORNOT W_4102  ; flag_assi_azzerati_pinza1
KEEP(011) W_6002  ; pinza1_in_ciclo

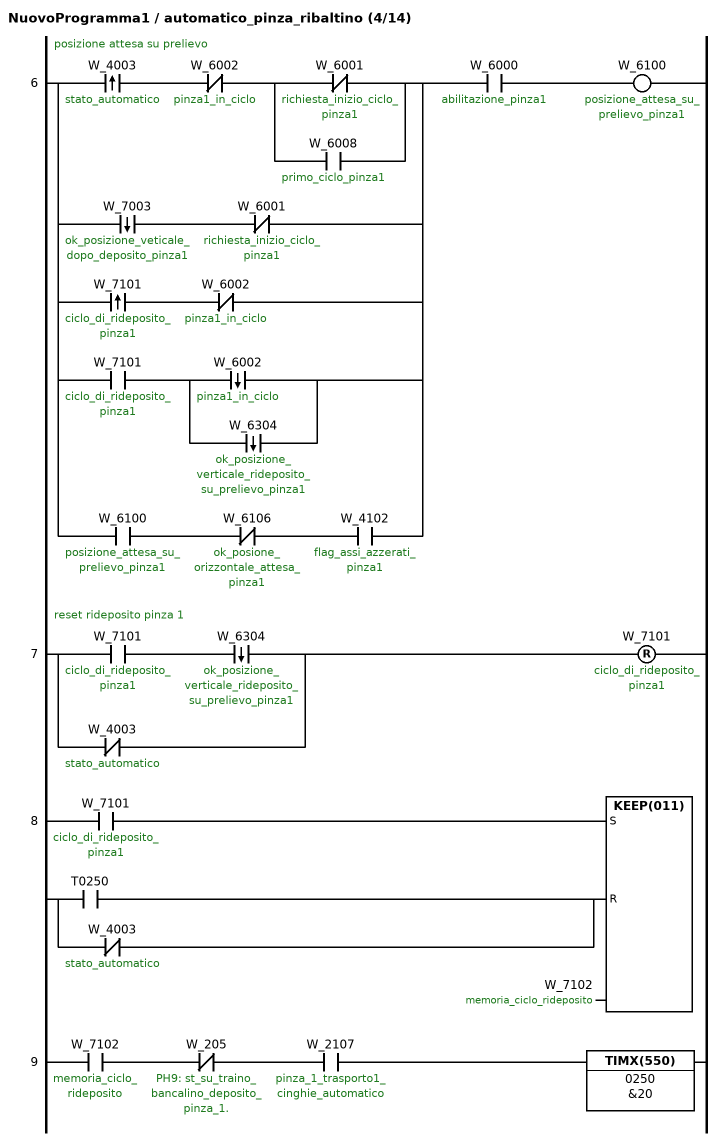
; rung 6: posizione attesa su prelievo
@LD W_4003  ; stato_automatico
ANDNOT W_6002  ; pinza1_in_ciclo
LDNOT W_6001  ; richiesta_inizio_ciclo_pinza1
OR W_6008  ; primo_ciclo_pinza1
ANDLD
%LD W_7003  ; ok_posizione_veticale_dopo_deposito_pinza1
ANDNOT W_6001  ; richiesta_inizio_ciclo_pinza1
ORLD
@LD W_7101  ; ciclo_di_rideposito_pinza1
ANDNOT W_6002  ; pinza1_in_ciclo
ORLD
LD W_7101  ; ciclo_di_rideposito_pinza1
%LD W_6002  ; pinza1_in_ciclo
%OR W_6304  ; ok_posizione_verticale_rideposito_su_prelievo_pinza1
ANDLD
ORLD
LD W_6100  ; posizione_attesa_su_prelievo_pinza1
ANDNOT W_6106  ; ok_posione_orizzontale_attesa_pinza1
AND W_4102  ; flag_assi_azzerati_pinza1
ORLD
AND W_6000  ; abilitazione_pinza1
OUT W_6100  ; posizione_attesa_su_prelievo_pinza1
; rung 7: reset rideposito pinza 1
LD W_7101  ; ciclo_di_rideposito_pinza1
%AND W_6304  ; ok_posizione_verticale_rideposito_su_prelievo_pinza1
ORNOT W_4003  ; stato_automatico
RSET W_7101  ; ciclo_di_rideposito_pinza1
; rung 8
LD W_7101  ; ciclo_di_rideposito_pinza1
LD T0250
ORNOT W_4003  ; stato_automatico
KEEP(011) W_7102  ; memoria_ciclo_rideposito
; rung 9
LD W_7102  ; memoria_ciclo_rideposito
ANDNOT W_205  ; PH9: st_su_traino_bancalino_deposito_pinza_1.
AND W_2107  ; pinza_1_trasporto1_cinghie_automatico
TIMX(550) 0250 &20

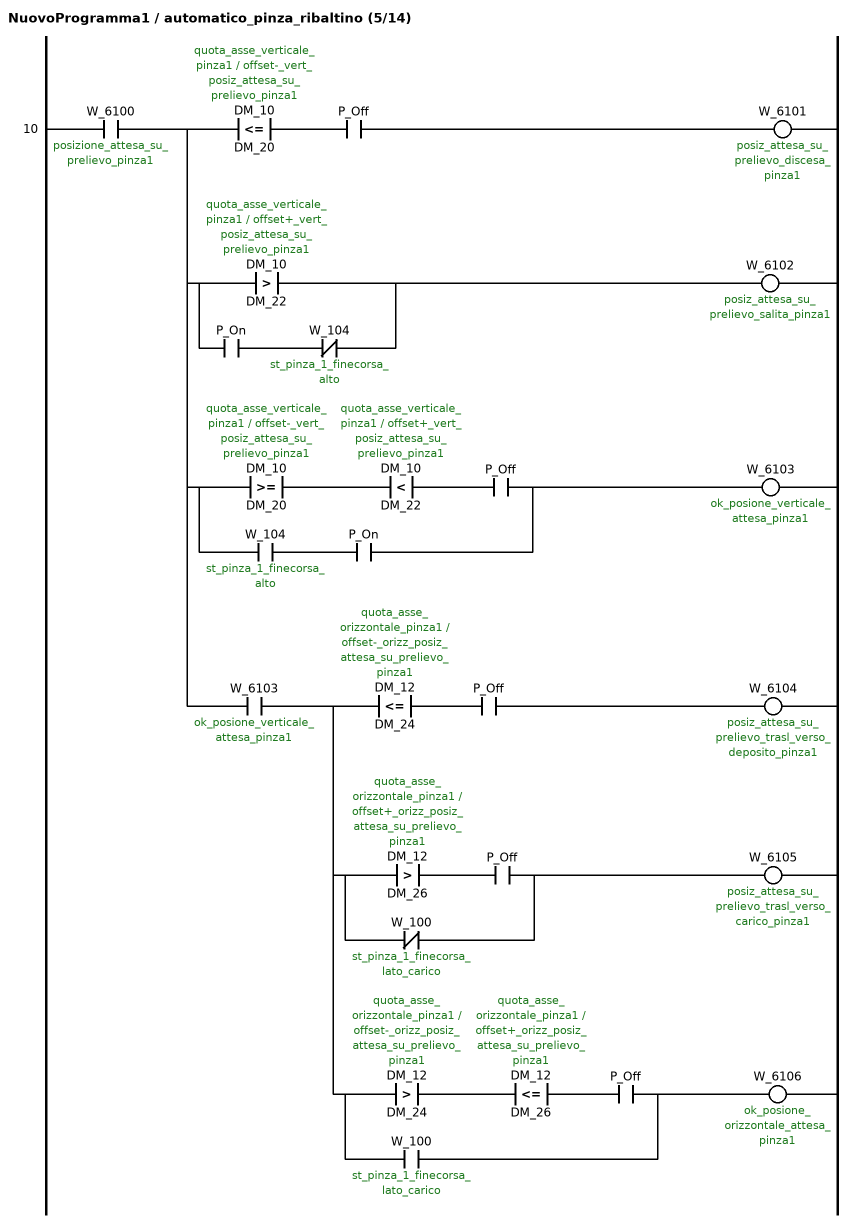
; rung 10
LD W_6100  ; posizione_attesa_su_prelievo_pinza1
OUT TR0
AND<=SL(318) DM_10 DM_20  ; quota_asse_verticale_pinza1, offset-_vert_posiz_attesa_su_prelievo_pinza1
AND P_Off
OUT W_6101  ; posiz_attesa_su_prelievo_discesa_pinza1
LD TR0
LD>SL(323) DM_10 DM_22  ; quota_asse_verticale_pinza1, offset+_vert_posiz_attesa_su_prelievo_pinza1
LD P_On
ANDNOT W_104  ; st_pinza_1_finecorsa_alto
ORLD
ANDLD
OUT W_6102  ; posiz_attesa_su_prelievo_salita_pinza1
LD TR0
LD>=SL(328) DM_10 DM_20  ; quota_asse_verticale_pinza1, offset-_vert_posiz_attesa_su_prelievo_pinza1
AND<SL(313) DM_10 DM_22  ; quota_asse_verticale_pinza1, offset+_vert_posiz_attesa_su_prelievo_pinza1
AND P_Off
LD W_104  ; st_pinza_1_finecorsa_alto
AND P_On
ORLD
ANDLD
OUT W_6103  ; ok_posione_verticale_attesa_pinza1
LD TR0
AND W_6103  ; ok_posione_verticale_attesa_pinza1
OUT TR0
AND<=SL(318) DM_12 DM_24  ; quota_asse_orizzontale_pinza1, offset-_orizz_posiz_attesa_su_prelievo_pinza1
AND P_Off
OUT W_6104  ; posiz_attesa_su_prelievo_trasl_verso_deposito_pinza1
LD TR0
LD>SL(323) DM_12 DM_26  ; quota_asse_orizzontale_pinza1, offset+_orizz_posiz_attesa_su_prelievo_pinza1
AND P_Off
ORNOT W_100  ; st_pinza_1_finecorsa_lato_carico
ANDLD
OUT W_6105  ; posiz_attesa_su_prelievo_trasl_verso_carico_pinza1
LD TR0
LD>SL(323) DM_12 DM_24  ; quota_asse_orizzontale_pinza1, offset-_orizz_posiz_attesa_su_prelievo_pinza1
AND<=SL(318) DM_12 DM_26  ; quota_asse_orizzontale_pinza1, offset+_orizz_posiz_attesa_su_prelievo_pinza1
AND P_Off
OR W_100  ; st_pinza_1_finecorsa_lato_carico
ANDLD
OUT W_6106  ; ok_posione_orizzontale_attesa_pinza1

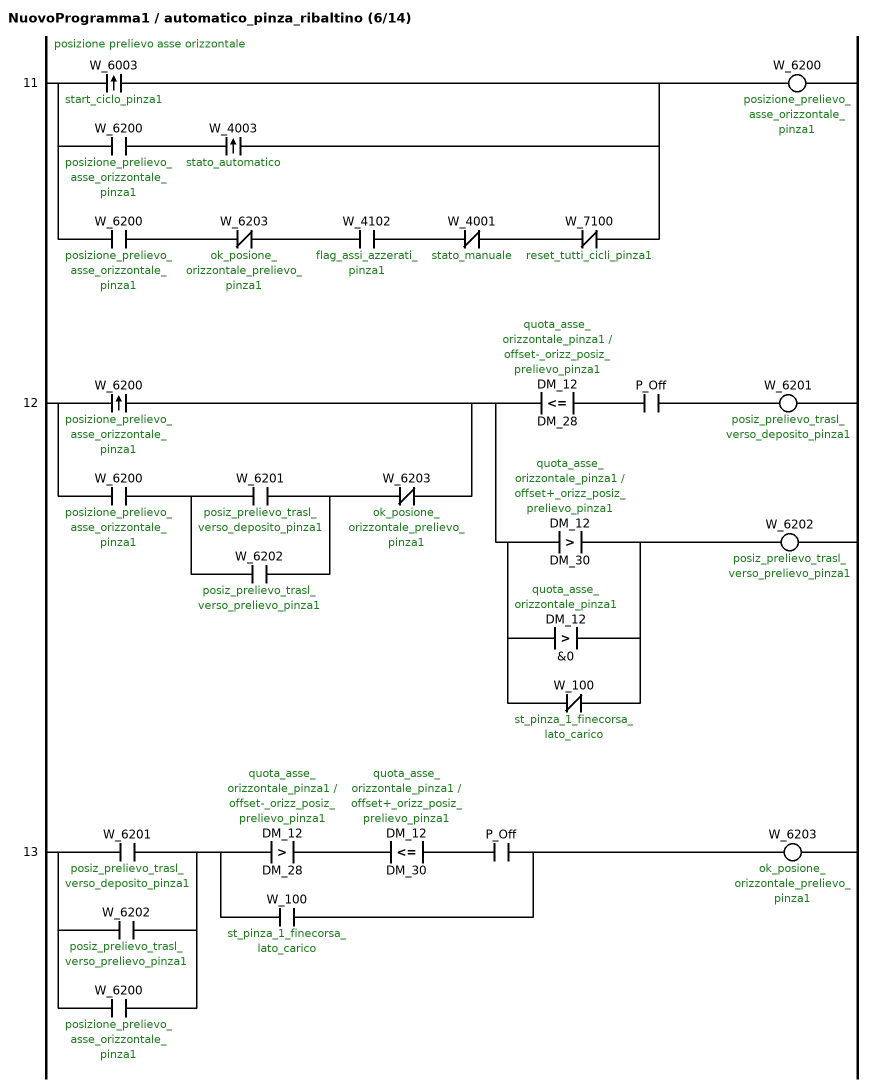
; rung 11: posizione prelievo asse orizzontale
@LD W_6003  ; start_ciclo_pinza1
LD W_6200  ; posizione_prelievo_asse_orizzontale_pinza1
@AND W_4003  ; stato_automatico
ORLD
LD W_6200  ; posizione_prelievo_asse_orizzontale_pinza1
ANDNOT W_6203  ; ok_posione_orizzontale_prelievo_pinza1
AND W_4102  ; flag_assi_azzerati_pinza1
ANDNOT W_4001  ; stato_manuale
ANDNOT W_7100  ; reset_tutti_cicli_pinza1
ORLD
OUT W_6200  ; posizione_prelievo_asse_orizzontale_pinza1
; rung 12
@LD W_6200  ; posizione_prelievo_asse_orizzontale_pinza1
LD W_6200  ; posizione_prelievo_asse_orizzontale_pinza1
LD W_6201  ; posiz_prelievo_trasl_verso_deposito_pinza1
OR W_6202  ; posiz_prelievo_trasl_verso_prelievo_pinza1
ANDLD
ANDNOT W_6203  ; ok_posione_orizzontale_prelievo_pinza1
ORLD
OUT TR0
AND<=SL(318) DM_12 DM_28  ; quota_asse_orizzontale_pinza1, offset-_orizz_posiz_prelievo_pinza1
AND P_Off
OUT W_6201  ; posiz_prelievo_trasl_verso_deposito_pinza1
LD TR0
LD>SL(323) DM_12 DM_30  ; quota_asse_orizzontale_pinza1, offset+_orizz_posiz_prelievo_pinza1
OR>SL(323) DM_12 &0  ; quota_asse_orizzontale_pinza1
ORNOT W_100  ; st_pinza_1_finecorsa_lato_carico
ANDLD
OUT W_6202  ; posiz_prelievo_trasl_verso_prelievo_pinza1
; rung 13
LD W_6201  ; posiz_prelievo_trasl_verso_deposito_pinza1
OR W_6202  ; posiz_prelievo_trasl_verso_prelievo_pinza1
OR W_6200  ; posizione_prelievo_asse_orizzontale_pinza1
LD>SL(323) DM_12 DM_28  ; quota_asse_orizzontale_pinza1, offset-_orizz_posiz_prelievo_pinza1
AND<=SL(318) DM_12 DM_30  ; quota_asse_orizzontale_pinza1, offset+_orizz_posiz_prelievo_pinza1
AND P_Off
OR W_100  ; st_pinza_1_finecorsa_lato_carico
ANDLD
OUT W_6203  ; ok_posione_orizzontale_prelievo_pinza1

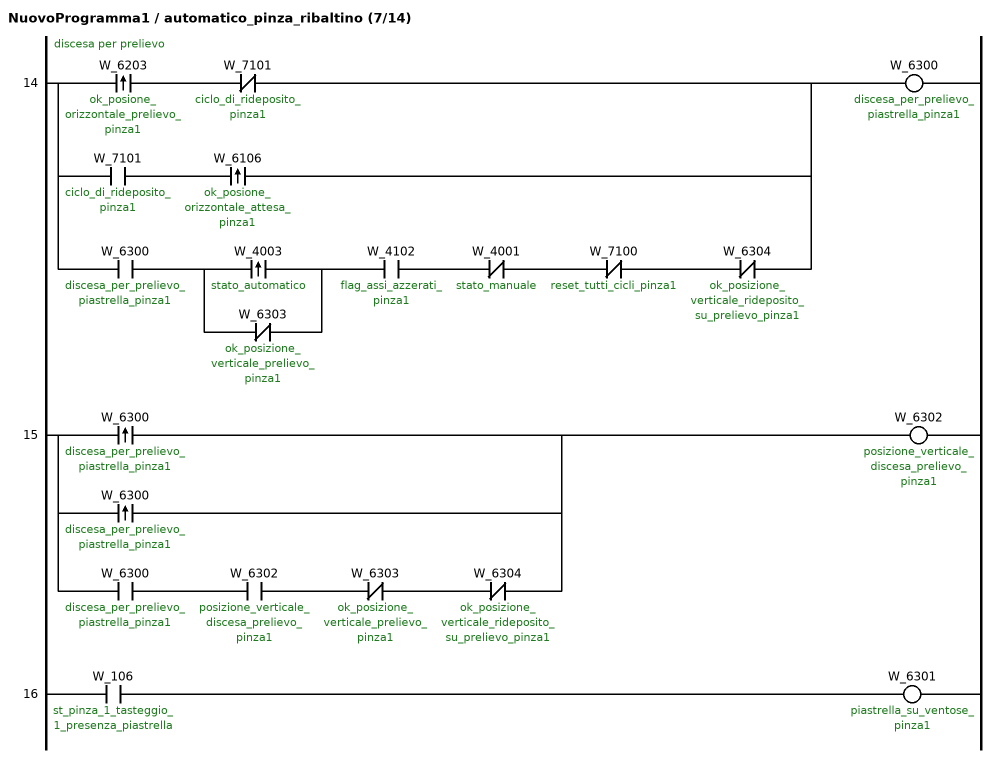
; rung 14: discesa per prelievo
@LD W_6203  ; ok_posione_orizzontale_prelievo_pinza1
ANDNOT W_7101  ; ciclo_di_rideposito_pinza1
LD W_7101  ; ciclo_di_rideposito_pinza1
@AND W_6106  ; ok_posione_orizzontale_attesa_pinza1
ORLD
LD W_6300  ; discesa_per_prelievo_piastrella_pinza1
@LD W_4003  ; stato_automatico
ORNOT W_6303  ; ok_posizione_verticale_prelievo_pinza1
ANDLD
AND W_4102  ; flag_assi_azzerati_pinza1
ANDNOT W_4001  ; stato_manuale
ANDNOT W_7100  ; reset_tutti_cicli_pinza1
ANDNOT W_6304  ; ok_posizione_verticale_rideposito_su_prelievo_pinza1
ORLD
OUT W_6300  ; discesa_per_prelievo_piastrella_pinza1
; rung 15
@LD W_6300  ; discesa_per_prelievo_piastrella_pinza1
@OR W_6300  ; discesa_per_prelievo_piastrella_pinza1
LD W_6300  ; discesa_per_prelievo_piastrella_pinza1
AND W_6302  ; posizione_verticale_discesa_prelievo_pinza1
ANDNOT W_6303  ; ok_posizione_verticale_prelievo_pinza1
ANDNOT W_6304  ; ok_posizione_verticale_rideposito_su_prelievo_pinza1
ORLD
OUT W_6302  ; posizione_verticale_discesa_prelievo_pinza1
; rung 16
LD W_106  ; st_pinza_1_tasteggio_1_presenza_piastrella
OUT W_6301  ; piastrella_su_ventose_pinza1

